(* IEC 61131-3 sources: types/src (part 2) *)

   END_TYPE

   TYPE EMHFDataRec147V1 : STRUCT
         version  : Byte := BYTE#1;   // Version
         resb1  : Byte;   // Reserved
         qualifierL1  : Word;   // Qualifier L1
         voltL1N  : Real;   // Voltage L1-N
         currentL1  : Real;   // Current L1
         apparentPowerL1  : Real;   // Apparent power L1
         activePowerL1  : Real;   // Active power L1
         reactivePowerQtotL1  : Real;   // Reactive power Qtot L1
         powerFactorL1  : Real;   // Power factor λ L1
         phaseAngleL1  : Real;   // Phase angle L1
         apparentEnergyLongL1  : LReal;   // Apparent energy L1
         totalActiveEnergyLongL1  : LReal;   // Active energy (total) L1
         totalReactiveEnergyLongL1  : LReal;   // Reactive energy (total) L1
         maxVoltL1N  : Real;   // Max. voltage L1-N
         maxCurrentL1  : Real;   // Max. current L1
         maxApparentPowerL1  : Real;   // Max. apparent power L1
         maxActivePowerL1  : Real;   // Max. active power L1
         maxReactivePowerQtotL1  : Real;   // Max. reactive power Qtot L1
         maxPowerFactorL1  : Real;   // Max. power factor λ L1
         minVoltL1N  : Real;   // Min. voltage L1-N
         minCurrentL1  : Real;   // Min. current L1
         minApparentPowerL1  : Real;   // Min. apparent power L1
         minActivePowerL1  : Real;   // Min. active power L1
         minReactivePowerQtotL1  : Real;   // Min. reactive power Qtot L1
         minPowerFactorL1  : Real;   // Min. power factor λ L1
         reactivePowerQnL1  : Real;   // Reactive power Qn L1
         voltL1Cycles10to12  : Real;   // Voltage L1 10-12 cycles
         currL1Cycles10to12  : Real;   // Current L1 10-12 cycles
         maxReactivePowerQnL1  : Real;   // Max. reactive power Qn L1
         minReactivePowerQnL1  : Real;   // Min. reactive power Qn L1
         fundVoltL1  : Real;   // Fundamental voltage L1
         fundCurrL1  : Real;   // Fundamental current L1
         fundApparentPowerL1  : Real;   // Fundamental apparent power L1
         fundReactivePowerL1  : Real;   // Fundamental reactive power L1
         fundActivePowerL1  : Real;   // Fundamental active power L1
         fundActiveFactorL1  : Real;   // Fundamental cos φ active factor L1
         maxFundVoltL1  : Real;   // Max. fundamental voltage L1
         maxFundCurrL1  : Real;   // Max. fundamental current L1
         maxFundApparentPowerL1  : Real;   // Max. fundamental apparent power L1
         maxFundReactivePowerL1  : Real;   // Max. fundamental reactive power L1
         maxFundActivePowerL1  : Real;   // Max. fundamental active power L1
         maxFundActiveFactorL1  : Real;   // Max. fundamental cos φ active factor L1
         minFundVoltL1  : Real;   // Min. fundamental voltage L1
         minFundCurrL1  : Real;   // Min. fundamental current L1
         minFundApparentPowerL1  : Real;   // Min. fundamental apparent power L1
         minFundReactivePowerL1  : Real;   // Min. fundamental reactive power L1
         minFundActivePowerL1  : Real;   // Min. fundamental active power L1
         minFundActiveFactorL1  : Real;   // Min. fundamental cos φ active factor L1
         tHDaNVoltL1  : Real;   // Total harmonic distortion (THD+N) voltage L1
         tHDaNCurrL1  : Real;   // Total harmonic distortion (THD+N) current L1
         maxTHDaNVoltL1  : Real;   // Max. total harmonic distortion (THD+N) voltage L1
         maxTHDaNCurrL1  : Real;   // Max. total harmonic distortion (THD+N) current L1
         minTHDaNVoltL1  : Real;   // Min. total harmonic distortion (THD+N) voltage L1
         minTHDaNCurrL1  : Real;   // Min. total harmonic distortion (THD+N) current L1
         voltDipValueL1  : Real;   // Voltage dip - value L1
         voltDipDurationL1  : Real;   // Voltage dip - duration L1
         voltSwellValueL1  : Real;   // Voltage swell - value L1
         voltSwellDurationL1  : Real;   // Voltage swell - duration L1
         voltPeakValueL1  : Real;   // Voltage peak value L1
         currPeakValueL1  : Real;   // Current peak value L1
         overCurrValueL1  : Real;   // Overcurrent value L1
      END_STRUCT;

   END_TYPE

   TYPE EMHFDataRec142V2 : STRUCT
         version  : Byte := BYTE#2;   // Version
         resb1  : Byte;   // Reserved
         voltL1N  : Real;   // Voltage L1-N
         voltL2N  : Real;   // Voltage L2-N
         voltL3N  : Real;   // Voltage L3-N
         voltL1L2  : Real;   // Voltage L1-L2
         voltL2L3  : Real;   // Voltage L2-L3
         voltL3L1  : Real;   // Voltage L3-L1
         currentL1  : Real;   // Current L1
         currentL2  : Real;   // Current L2
         currentL3  : Real;   // Current L3
         powerFactorL1  : Real;   // Power factor λ L1
         powerFactorL2  : Real;   // Power factor λ L2
         powerFactorL3  : Real;   // Power factor λ L3
         powerFactorL1L2L3  : Real;   // Power factor λ L1 L2 L3
         frequencyL1L2L3  : Real;   // Frequency L1 L2 L3
         amplUnbalanceVolt  : Real;   // Amplitude unbalance voltage U2
         amplUnbalanceCurrent  : Real;   // Amplitude unbalance current Iasym
         apparentPowerL1  : Real;   // Apparent power L1
         apparentPowerL2  : Real;   // Apparent power L2
         apparentPowerL3  : Real;   // Apparent power L3
         apparentPowerL1L2L3  : Real;   // Apparent power L1 L2 L3
         reactivePowerQtotL1  : Real;   // Reactive power Qtot L1
         reactivePowerQtotL2  : Real;   // Reactive power Qtot L2
         reactivePowerQtotL3  : Real;   // Reactive power Qtot L3
         reactivePowerQtotL1L2L3  : Real;   // Reactive power Qtot L1 L2 L3
         activePowerL1  : Real;   // Active power L1
         activePowerL2  : Real;   // Active power L2
         activePowerL3  : Real;   // Active power L3
         activePowerL1L2L3  : Real;   // Active power L1 L2 L3
         phaseAngleL1  : Real;   // Phase angle L1
         phaseAngleL2  : Real;   // Phase angle L2
         phaseAngleL3  : Real;   // Phase angle L3
         apparentEnergyL1L2L3  : Real;   // Apparent energy L1 L2 L3
         totalReactiveEnergyL1L2L3  : Real;   // Total reactive energy L1 L2 L3
         totalActiveEnergyL1L2L3  : Real;   // Total active energy L1 L2 L3
         reactiveEnergyInL1L2L3  : Real;   // Reactive energy inflow L1 L2 L3
         reactiveEnergyOutL1L2L3  : Real;   // Reactive energy outflow L1 L2 L3
         activeEnergyInL1L2L3  : Real;   // Active energy inflow L1 L2 L3
         activeEnergyOutL1L2L3  : Real;   // Active energy outflow L1 L2 L3
         apparentEnergyLongL1L2L3  : LReal;   // Apparent energy L1 L2 L3
         totalReactiveEnergyLongL1L2L3  : LReal;   // Total reactive energy L1 L2 L3
         totalActiveEnergyLongL1L2L3  : LReal;   // Total active energy L1 L2 L3
         reactiveEnergyInLongL1L2L3  : LReal;   // Reactive energy inflow L1 L2 L3
         reactiveEnergyOutLongL1L2L3  : LReal;   // Reactive energy outflow L1 L2 L3
         activeEnergyInLongL1L2L3  : LReal;   // Active energy inflow L1 L2 L3
         activeEnergyOutLongL1L2L3  : LReal;   // Active energy outflow L1 L2 L3
         neutralCurrentIn  : Real;   // Neutral current IN
      END_STRUCT;

   END_TYPE

   TYPE EMHFDataRec148V1 : STRUCT
         version  : Byte := BYTE#1;   // Version
         resb1  : Byte;   // Reserved
         qualifierL2  : Word;   // Qualifier L2
         voltL2N  : Real;   // Voltage L2-N
         currentL2  : Real;   // Current L2
         apparentPowerL2  : Real;   // Apparent power L2
         activePowerL2  : Real;   // Active power L2
         reactivePowerQtotL2  : Real;   // Reactive power Qtot L2
         powerFactorL2  : Real;   // Power factor λ L2
         phaseAngleL2  : Real;   // Phase angle L2
         apparentEnergyLongL2  : LReal;   // Apparent energy L2
         totalActiveEnergyLongL2  : LReal;   // Active energy (total) L2
         totalReactiveEnergyLongL2  : LReal;   // Reactive energy (total) L2
         maxVoltL2N  : Real;   // Max. voltage L2-N
         maxCurrentL2  : Real;   // Max. current L2
         maxApparentPowerL2  : Real;   // Max. apparent power L2
         maxActivePowerL2  : Real;   // Max. active power L2
         maxReactivePowerQtotL2  : Real;   // Max. reactive power Qtot L2
         maxPowerFactorL2  : Real;   // Max. power factor λ L2
         minVoltL2N  : Real;   // Min. voltage L2-N
         minCurrentL2  : Real;   // Min. current L2
         minApparentPowerL2  : Real;   // Min. apparent power L2
         minActivePowerL2  : Real;   // Min. active power L2
         minReactivePowerQtotL2  : Real;   // Min. reactive power Qtot L2
         minPowerFactorL2  : Real;   // Min. power factor λ L2
         reactivePowerQnL2  : Real;   // Reactive power Qn L2
         voltL2Cycles10to12  : Real;   // Voltage L2 10-12 cycles
         currL2Cycles10to12  : Real;   // Current L2 10-12 cycles
         maxReactivePowerQnL2  : Real;   // Max. reactive power Qn L2
         minReactivePowerQnL2  : Real;   // Min. reactive power Qn L2
         fundVoltL2  : Real;   // Fundamental voltage L2
         fundCurrL2  : Real;   // Fundamental current L2
         fundApparentPowerL2  : Real;   // Fundamental apparent power L2
         fundReactivePowerL2  : Real;   // Fundamental reactive power L2
         fundActivePowerL2  : Real;   // Fundamental active power L2
         fundActiveFactorL2  : Real;   // Fundamental cos φ active factor L2
         maxFundVoltL2  : Real;   // Max. fundamental voltage L2
         maxFundCurrL2  : Real;   // Max. fundamental current L2
         maxFundApparentPowerL2  : Real;   // Max. fundamental apparent power L2
         maxFundReactivePowerL2  : Real;   // Max. fundamental reactive power L2
         maxFundActivePowerL2  : Real;   // Max. fundamental active power L2
         maxFundActiveFactorL2  : Real;   // Max. fundamental cos φ active factor L2
         minFundVoltL2  : Real;   // Min. fundamental voltage L2
         minFundCurrL2  : Real;   // Min. fundamental current L2
         minFundApparentPowerL2  : Real;   // Min. fundamental apparent power L2
         minFundReactivePowerL2  : Real;   // Min. fundamental reactive power L2
         minFundActivePowerL2  : Real;   // Min. fundamental active power L2
         minFundActiveFactorL2  : Real;   // Min. fundamental cos φ active factor L2
         tHDaNVoltL2  : Real;   // Total harmonic distortion (THD+N) voltage L2
         tHDaNCurrL2  : Real;   // Total harmonic distortion (THD+N) current L2
         maxTHDaNVoltL2  : Real;   // Max. total harmonic distortion (THD+N) voltage L2
         maxTHDaNCurrL2  : Real;   // Max. total harmonic distortion (THD+N) current L2
         minTHDaNVoltL2  : Real;   // Min. total harmonic distortion (THD+N) voltage L2
         minTHDaNCurrL2  : Real;   // Min. total harmonic distortion (THD+N) current L2
         voltDipValueL2  : Real;   // Voltage dip - value L2
         voltDipDurationL2  : Real;   // Voltage dip - duration L2
         voltSwellValueL2  : Real;   // Voltage swell - value L2
         voltSwellDurationL2  : Real;   // Voltage swell - duration L2
         voltPeakValueL2  : Real;   // Voltage peak value L2
         currPeakValueL2  : Real;   // Current peak value L2
         overCurrValueL2  : Real;   // Overcurrent value L2
      END_STRUCT;

   END_TYPE

   TYPE EMSTDataRec142V2 : STRUCT
         version  : Byte := BYTE#2;   // Version
         resb1  : Byte;   // Reserved
         voltL1N  : Real;   // Voltage L1-N
         voltL2N  : Real;   // Voltage L2-N
         voltL3N  : Real;   // Voltage L3-N
         voltL1L2  : Real;   // Voltage L1-L2
         voltL2L3  : Real;   // Voltage L2-L3
         voltL3L1  : Real;   // Voltage L3-L1
         currentL1  : Real;   // Current L1
         currentL2  : Real;   // Current L2
         currentL3  : Real;   // Current L3
         powerFactorL1  : Real;   // Power factor λ L1
         powerFactorL2  : Real;   // Power factor λ L2
         powerFactorL3  : Real;   // Power factor λ L3
         powerFactorL1L2L3  : Real;   // Power factor L1 L2 L3
         frequencyL1L2L3  : Real;   // Frequency L1 L2 L3
         amplUnbalanceVolt  : Real;   // Amplitude unbalance voltage U2
         amplUnbalanceCurrent  : Real;   // Amplitude unbalance current Iasym
         apparentPowerL1  : Real;   // Apparent power L1
         apparentPowerL2  : Real;   // Apparent power L2
         apparentPowerL3  : Real;   // Apparent power L3
         apparentPowerL1L2L3  : Real;   // Apparent power L1 L2 L3
         reactivePowerQtotL1  : Real;   // Reactive power Qtot L1
         reactivePowerQtotL2  : Real;   // Reactive power Qtot L2
         reactivePowerQtotL3  : Real;   // Reactive power Qtot L3
         reactivePowerQtotL1L2L3  : Real;   // Reactive power Qtot L1 L2 L3
         activePowerL1  : Real;   // Active power L1
         activePowerL2  : Real;   // Active power L2
         activePowerL3  : Real;   // Active power L3
         activePowerL1L2L3  : Real;   // Active power L1 L2 L3
         phaseAngleL1  : Real;   // Phase angle L1
         phaseAngleL2  : Real;   // Phase angle L2
         phaseAngleL3  : Real;   // Phase angle L3
         apparentEnergyL1L2L3  : Real;   // Apparent energy L1 L2 L3
         totalReactiveEnergyL1L2L3  : Real;   // Total reactive energy L1 L2 L3
         totalActiveEnergyL1L2L3  : Real;   // Total active energy L1 L2 L3
         reactiveEnergyInL1L2L3  : Real;   // Reactive energy inflow L1 L2 L3
         reactiveEnergyOutL1L2L3  : Real;   // Reactive energy outflow L1 L2 L3
         activeEnergyInL1L2L3  : Real;   // Active energy inflow L1 L2 L3
         activeEnergyOutL1L2L3  : Real;   // Active energy outflow L1 L2 L3
         apparentEnergyLongL1L2L3  : LReal;   // Apparent energy L1 L2 L3
         totalReactiveEnergyLongL1L2L3  : LReal;   // Total reactive energy L1 L2 L3
         totalActiveEnergyLongL1L2L3  : LReal;   // Total active energy L1 L2 L3
         reactiveEnergyInLongL1L2L3  : LReal;   // Reactive energy inflow L1 L2 L3
         reactiveEnergyOutLongL1L2L3  : LReal;   // Reactive energy outflow L1 L2 L3
         activeEnergyInLongL1L2L3  : LReal;   // Active energy inflow L1 L2 L3
         activeEnergyOutLongL1L2L3  : LReal;   // Active energy outflow L1 L2 L3
         neutralCurrentIn  : Real;   // Neutral current IN
      END_STRUCT;

   END_TYPE

   TYPE EMHFDataRec154 : STRUCT
         version  : Byte := BYTE#2;   // Version
         resb1  : Byte;   // Reserved
         maxVoltL1N  : RealValueAndPNIOTimeStamp;   // Max. voltage L1-N
         maxVoltL2N  : RealValueAndPNIOTimeStamp;   // Max. voltage L2-N
         maxVoltL3N  : RealValueAndPNIOTimeStamp;   // Max. voltage L3-N
         maxVoltL1L2  : RealValueAndPNIOTimeStamp;   // Max. voltage L1-L2
         maxVoltL2L3  : RealValueAndPNIOTimeStamp;   // Max. voltage L2-L3
         maxVoltL3L1  : RealValueAndPNIOTimeStamp;   // Max. voltage L3-L1
         maxCurrentL1  : RealValueAndPNIOTimeStamp;   // Max. current L1
         maxCurrentL2  : RealValueAndPNIOTimeStamp;   // Max. current L2
         maxCurrentL3  : RealValueAndPNIOTimeStamp;   // Max. current L3
         maxApparentPowerL1  : RealValueAndPNIOTimeStamp;   // Max. apparent power L1
         maxApparentPowerL2  : RealValueAndPNIOTimeStamp;   // Max. apparent power L2
         maxApparentPowerL3  : RealValueAndPNIOTimeStamp;   // Max. apparent power L3
         maxActivePowerL1  : RealValueAndPNIOTimeStamp;   // Max. active power L1
         maxActivePowerL2  : RealValueAndPNIOTimeStamp;   // Max. active power L2
         maxActivePowerL3  : RealValueAndPNIOTimeStamp;   // Max. active power L3
         maxReactivePowerQtotL1  : RealValueAndPNIOTimeStamp;   // Max. reactive power Qtot L1
         maxReactivePowerQtotL2  : RealValueAndPNIOTimeStamp;   // Max. reactive power Qtot L2
         maxReactivePowerQtotL3  : RealValueAndPNIOTimeStamp;   // Max. reactive power Qtot L3
         maxPowerFactorL1  : RealValueAndPNIOTimeStamp;   // Max. power factor λ L1
         maxPowerFactorL2  : RealValueAndPNIOTimeStamp;   // Max. power factor λ L2
         maxPowerFactorL3  : RealValueAndPNIOTimeStamp;   // Max. power factor λ L3
         maxFrequency  : RealValueAndPNIOTimeStamp;   // Max. frequency
         maxApparentPowerL1L2L3  : RealValueAndPNIOTimeStamp;   // Max. apparent power L1 L2 L3
         maxActivePowerL1L2L3  : RealValueAndPNIOTimeStamp;   // Max. active power L1 L2 L3
         maxReactivePowerQtotL1L2L3  : RealValueAndPNIOTimeStamp;   // Max. reactive power Qtot L1 L2 L3
         maxPowerFactorL1L2L3  : RealValueAndPNIOTimeStamp;   // Max. power factor λ L1L2L3
         maxReactivePowerQnL1  : RealValueAndPNIOTimeStamp;   // Max. reactive power Qn L1
         maxReactivePowerQnL2  : RealValueAndPNIOTimeStamp;   // Max. reactive power Qn L2
         maxReactivePowerQnL3  : RealValueAndPNIOTimeStamp;   // Max. reactive power Qn L3
         maxMeanVoltLN  : RealValueAndPNIOTimeStamp;   // Max. mean voltage L-N
         maxMeanVoltLL  : RealValueAndPNIOTimeStamp;   // Max. mean voltage L-L
         maxSumMeanCurrL1L2L3  : RealValueAndPNIOTimeStamp;   // Max. sum mean value current L1L2L3
         maxFundVoltL1  : RealValueAndPNIOTimeStamp;   // Max. fundamental voltage L1
         maxFundVoltL2  : RealValueAndPNIOTimeStamp;   // Max. fundamental voltage L2
         maxFundVoltL3  : RealValueAndPNIOTimeStamp;   // Max. fundamental voltage L3
         maxFundCurrL1  : RealValueAndPNIOTimeStamp;   // Max. fundamental current L1
         maxFundCurrL2  : RealValueAndPNIOTimeStamp;   // Max. fundamental current L2
         maxFundCurrL3  : RealValueAndPNIOTimeStamp;   // Max. fundamental current L3
         maxFundApparentPowerL1  : RealValueAndPNIOTimeStamp;   // Max. fundamental apparent power L1
         maxFundApparentPowerL2  : RealValueAndPNIOTimeStamp;   // Max. fundamental apparent power L2
         maxFundApparentPowerL3  : RealValueAndPNIOTimeStamp;   // Max. fundamental apparent power L3
         maxFundReactivePowerL1  : RealValueAndPNIOTimeStamp;   // Max. fundamental reactive power L1
         maxFundReactivePowerL2  : RealValueAndPNIOTimeStamp;   // Max. fundamental reactive power L2
         maxFundReactivePowerL3  : RealValueAndPNIOTimeStamp;   // Max. fundamental reactive power L3
         maxFundActivePowerL1  : RealValueAndPNIOTimeStamp;   // Max. fundamental active power L1
         maxFundActivePowerL2  : RealValueAndPNIOTimeStamp;   // Max. fundamental active power L2
         maxFundActivePowerL3  : RealValueAndPNIOTimeStamp;   // Max. fundamental active power L3
         maxFundActiveFactorL1  : RealValueAndPNIOTimeStamp;   // Max. fundamental cos φ active factor L1
         maxFundActiveFactorL2  : RealValueAndPNIOTimeStamp;   // Max. fundamental cos φ active factor L2
         maxFundActiveFactorL3  : RealValueAndPNIOTimeStamp;   // Max. fundamental cos φ active factor L3
         maxTHDaNVoltL1  : RealValueAndPNIOTimeStamp;   // Max. total harmonic distortion (THD+N) voltage L1
         maxTHDaNVoltL2  : RealValueAndPNIOTimeStamp;   // Max. total harmonic distortion (THD+N) voltage L2
         maxTHDaNVoltL3  : RealValueAndPNIOTimeStamp;   // Max. total harmonic distortion (THD+N) voltage L3
         maxTHDaNCurrL1  : RealValueAndPNIOTimeStamp;   // Max. total harmonic distortion (THD+N) current L1
         maxTHDaNCurrL2  : RealValueAndPNIOTimeStamp;   // Max. total harmonic distortion (THD+N) current L2
         maxTHDaNCurrL3  : RealValueAndPNIOTimeStamp;   // Max. total harmonic distortion (THD+N) current L3
         maxNeutralCurr  : RealValueAndPNIOTimeStamp;   // Max. neutral current
      END_STRUCT;

   END_TYPE

   TYPE EMSTDataRec143 : STRUCT
         version  : Byte := BYTE#1;   // Version
         resb1  : Byte;   // Reserved
         controlStatusByte1L1  : Byte;   // Status / control byte 1 - L1
         controlStatusByte2L1  : Byte;   // Status / control byte 2 - L1
         controlStatusByte1L2  : Byte;   // Status / control byte 1 - L2
         controlStatusByte2L2  : Byte;   // Status / control byte 2 - L2
         controlStatusByte1L3  : Byte;   // Status / control byte 1 - L3
         controlStatusByte2L3  : Byte;   // Status / control byte 2 - L3
         activeEnergyInLongL1  : LReal;   // Active energy inflow (initial value) L1
         activeEnergyOutLongL1  : LReal;   // Active energy outflow (initial value) L1
         reactiveEnergyInLongL1  : LReal;   // Reactive energy inflow (initial value) L1
         reactiveEnergyOutLongL1  : LReal;   // Reactive energy outflow (initial value) L1
         apparentEnergyLongL1  : LReal;   // Apparent energy (initial value) L1
         activeEnergyInLongL2  : LReal;   // Active energy inflow (initial value) L2
         activeEnergyOutLongL2  : LReal;   // Active energy outflow (initial value) L2
         reactiveEnergyInLongL2  : LReal;   // Reactive energy inflow (initial value) L2
         reactiveEnergyOutLongL2  : LReal;   // Reactive energy outflow (initial value) L2
         apparentEnergyLongL2  : LReal;   // Apparent energy (initial value) L2
         activeEnergyInLongL3  : LReal;   // Active energy inflow (initial value) L3
         activeEnergyOutLongL3  : LReal;   // Active energy outflow (initial value) L3
         reactiveEnergyInLongL3  : LReal;   // Reactive energy inflow (initial value) L3
         reactiveEnergyOutLongL3  : LReal;   // Reactive energy outflow (initial value) L3
         apparentEnergyLongL3  : LReal;   // Apparent energy (initial value) L3
         ovCntActiveEnergyInL1  : UInt;   // Overflow counter active energy inflow L1
         ovCntActiveEnergyOutL1  : UInt;   // Overflow counter active energy outflow L1
         ovCntReactiveEnergyInL1  : UInt;   // Overflow counter reactive energy inflow L1
         ovCntReactiveEnergyOutL1  : UInt;   // Overflow counter reactive energy outflow L1
         ovCntApparentEnergyL1  : UInt;   // Overflow counter apparent energy L1
         ovCntActiveEnergyInL2  : UInt;   // Overflow counter active energy inflow L2
         ovCntActiveEnergyOutL2  : UInt;   // Overflow counter active energy outflow L2
         ovCntReactiveEnergyInL2  : UInt;   // Overflow counter reactive energy inflow L2
         ovCntReactiveEnergyOutL2  : UInt;   // Overflow counter reactive energy outflow L2
         ovCntApparentEnergyL2  : UInt;   // Overflow counter apparent energy L2
         ovCntActiveEnergyInL3  : UInt;   // Overflow counter active energy inflow L3
         ovCntActiveEnergyOutL3  : UInt;   // Overflow counter active energy outflow L3
         ovCntReactiveEnergyInL3  : UInt;   // Overflow counter reactive energy inflow L3
         ovCntReactiveEnergyOutL3  : UInt;   // Overflow counter reactive energy outflow L3
         ovCntApparentEnergyL3  : UInt;   // Overflow counter apparent energy L3
         operHoursCntL1  : Real;   // Operating hours counter L1 (initial value)
         operHoursCntL2  : Real;   // Operating hours counter L2 (initial value)
         operHoursCntL3  : Real;   // Operating hours counter L3 (initial value)
      END_STRUCT;

   END_TYPE

   TYPE EMSTDataRec135 : STRUCT
         majMinVer  : Byte := BYTE#0;   // Major / minor version
         dataRecordNum  : Byte := BYTE#151;   // Data record number for data record mapping = 151
         numMeasValues  : Byte := BYTE#150;   // Number of measured values for data record mapping
         resb3  : Byte;   // Reserved
         measValueID  : Array[1..150] of Word;   // ID of measured value for data record mapping
      END_STRUCT;

   END_TYPE

   TYPE EMHFDataRec149V1 : STRUCT
         version  : Byte := BYTE#1;   // Version
         resb1  : Byte;   // Reserved
         qualifierL3  : Word;   // Qualifier L3
         voltL3N  : Real;   // Voltage L3-N
         currentL3  : Real;   // Current L3
         apparentPowerL3  : Real;   // Apparent power L3
         activePowerL3  : Real;   // Active power L3
         reactivePowerQtotL3  : Real;   // Reactive power Qtot L3
         powerFactorL3  : Real;   // Power factor λ L3
         phaseAngleL3  : Real;   // Phase angle L3
         apparentEnergyLongL3  : LReal;   // Apparent energy L3
         totalActiveEnergyLongL3  : LReal;   // Active energy (total) L3
         totalReactiveEnergyLongL3  : LReal;   // Reactive energy (total) L3
         maxVoltL3N  : Real;   // Max. voltage L3-N
         maxCurrentL3  : Real;   // Max. current L3
         maxApparentPowerL3  : Real;   // Max. apparent power L3
         maxActivePowerL3  : Real;   // Max. active power L3
         maxReactivePowerQtotL3  : Real;   // Max. reactive power Qtot L3
         maxPowerFactorL3  : Real;   // Max. power factor λ L3
         minVoltL3N  : Real;   // Min. voltage L3-N
         minCurrentL3  : Real;   // Min. current L3
         minApparentPowerL3  : Real;   // Min. apparent power L3
         minActivePowerL3  : Real;   // Min. active power L3
         minReactivePowerQtotL3  : Real;   // Min. reactive power Qtot L3
         minPowerFactorL3  : Real;   // Min. power factor λ L3
         reactivePowerQnL3  : Real;   // Reactive power Qn L3
         voltL3Cycles10to12  : Real;   // Voltage L3 10-12 cycles
         currL3Cycles10to12  : Real;   // Current L3 10-12 cycles
         maxReactivePowerQnL3  : Real;   // Max. reactive power Qn L3
         minReactivePowerQnL3  : Real;   // Min. reactive power Qn L3
         fundVoltL3  : Real;   // Fundamental voltage L3
         fundCurrL3  : Real;   // Fundamental current L3
         fundApparentPowerL3  : Real;   // Fundamental apparent power L3
         fundReactivePowerL3  : Real;   // Fundamental reactive power L3
         fundActivePowerL3  : Real;   // Fundamental active power L3
         fundActiveFactorL3  : Real;   // Fundamental cos φ active factor L3
         maxFundVoltL3  : Real;   // Max. fundamental voltage L3
         maxFundCurrL3  : Real;   // Max. fundamental current L3
         maxFundApparentPowerL3  : Real;   // Max. fundamental apparent power L3
         maxFundReactivePowerL3  : Real;   // Max. fundamental reactive power L3
         maxFundActivePowerL3  : Real;   // Max. fundamental active power L3
         maxFundActiveFactorL3  : Real;   // Max. fundamental cos φ active factor L3
         minFundVoltL3  : Real;   // Min. fundamental voltage L3
         minFundCurrL3  : Real;   // Min. fundamental current L3
         minFundApparentPowerL3  : Real;   // Min. fundamental apparent power L3
         minFundReactivePowerL3  : Real;   // Min. fundamental reactive power L3
         minFundActivePowerL3  : Real;   // Min. fundamental active power L3
         minFundActiveFactorL3  : Real;   // Min. fundamental cos φ active factor L3
         tHDaNVoltL3  : Real;   // Total harmonic distortion (THD+N) voltage L3
         tHDaNCurrL3  : Real;   // Total harmonic distortion (THD+N) current L3
         maxTHDaNVoltL3  : Real;   // Max. total harmonic distortion (THD+N) voltage L3
         maxTHDaNCurrL3  : Real;   // Max. total harmonic distortion (THD+N) current L3
         minTHDaNVoltL3  : Real;   // Min. total harmonic distortion (THD+N) voltage L3
         minTHDaNCurrL3  : Real;   // Min. total harmonic distortion (THD+N) current L3
         voltDipValueL3  : Real;   // Voltage dip - value L3
         voltDipDurationL3  : Real;   // Voltage dip - duration L3
         voltSwellValueL3  : Real;   // Voltage swell - value L3
         voltSwellDurationL3  : Real;   // Voltage swell - duration L3
         voltPeakValueL3  : Real;   // Voltage peak value L3
         currPeakValueL3  : Real;   // Current peak value L3
         overCurrValueL3  : Real;   // Overcurrent value L3
      END_STRUCT;

   END_TYPE

   TYPE EMHFDataRec150V1 : STRUCT
         version  : Byte := BYTE#1;   // Version
         resb1  : Byte;   // Reserved
         operHoursCntL1L2L3  : Real;   // Operating hours counter L1 L2 L3
         operHoursCntL1  : Real;   // Operating hours counter L1
         operHoursCntL2  : Real;   // Operating hours counter L2
         operHoursCntL3  : Real;   // Operating hours counter L3
         statusLimViolGW1to16  : Word;   // Status limit violation GW 1...16
         statusEnergyCntOv  : Word;   // Status of energy counter overflows
         cntLimViolGw1  : UDInt;   // Counter limit violation GW 1
         cntLimViolGw2  : UDInt;   // Counter limit violation GW 2
         cntLimViolGw3  : UDInt;   // Counter limit violation GW 3
         cntLimViolGw4  : UDInt;   // Counter limit violation GW 4
         cntLimViolGw5  : UDInt;   // Counter limit violation GW 5
         cntLimViolGw6  : UDInt;   // Counter limit violation GW 6
         cntLimViolGw7  : UDInt;   // Counter limit violation GW 7
         cntLimViolGw8  : UDInt;   // Counter limit violation GW 8
         cntLimViolGw9  : UDInt;   // Counter limit violation GW 9
         cntLimViolGw10  : UDInt;   // Counter limit violation GW 10
         cntLimViolGw11  : UDInt;   // Counter limit violation GW 11
         cntLimViolGw12  : UDInt;   // Counter limit violation GW 12
         cntLimViolGw13  : UDInt;   // Counter limit violation GW 13
         cntLimViolGw14  : UDInt;   // Counter limit violation GW 14
         cntLimViolGw15  : UDInt;   // Counter limit violation GW 15
         cntLimViolGw16  : UDInt;   // Counter limit violation GW 16
         qualifierL1L2L3  : Word;   // Qualifier L1 L2 L3
         powerQualityAnalysis  : UDInt;   // Power quality analysis - Qualifier
         currentModuleTime  : PNIOTimeStamp;   // Current module time
      END_STRUCT;

   END_TYPE

   TYPE TMTimerDIDQ10DataRec : STRUCT
         majMinVer  : Byte := BYTE#1;   // Major / minor version
         channelParamLength  : Byte := BYTE#36;   // Length of the parameter data = 36
         reserved0  : Word;   // Reserved
         pwmPeriod  : Byte;   // Reserved/ PWM period for the digital outputs
         enableDiagnostics  : Byte;   // Enable diagnostics / Reaction to CPU STOP
         reserved1  : Word;   // Reserved
         operatingModeDI0  : Byte;   // Reserved / invert input signal / operating mode DI0
         inputDelayDI0  : Byte;   // Reserved / Input delay / Filter frequency DI0
         operatingModeDI1  : Byte;   // Reserved / invert input signal / operating mode DI1
         inputDelayDI1  : Byte;   // Reserved / Input delay / Filter frequency DI1
         operatingModeDI2  : Byte;   // Reserved / invert input signal / HW enable with DI3 / operating mode DI2
         inputDelayDI2  : Byte;   // Reserved / Input delay / Filter frequency DI2
         operatingModeDI3  : Byte;   // Reserved / invert input signal / operating mode DI1
         inputDelayDI3  : Byte;   // Reserved / Input delay DI3
         operatingModeDQ0  : Byte;   // High-speed output / Substitute value / invert input signal / HW enable / operating mode DQ0
         reserved2  : Byte;   // Reserved
         operatingModeDQ1  : Byte;   // High-speed output / Substitute value / invert input signal / HW enable / operating mode DQ1
         reserved3  : Byte;   // Reserved
         operatingModeDQ2  : Byte;   // High-speed output / Substitute value / invert input signal / HW enable / operating mode DQ2
         reserved4  : Byte;   // Reserved
         operatingModeDQ3  : Byte;   // High-speed output / Substitute value / invert input signal / Reserved / operating mode DQ3
         reserved5  : Byte;   // Reserved
         operatingModeDQ4  : Byte;   // High-speed output / Substitute value / invert input signal / Reserved / operating mode DQ4
         reserved6  : Byte;   // Reserved
         operatingModeDQ5  : Byte;   // High-speed output / Substitute value / invert input signal / Reserved / operating mode DQ5
         reserved7  : Byte;   // Reserved
         reserved8  : DWord;   // Reserved
         reserved9  : DWord;   // Reserved
         reserved10  : DWord;   // Reserved
      END_STRUCT;

   END_TYPE

   TYPE EMSTDataRec130 : STRUCT
         majMinVer  : Byte := BYTE#0;   // Major / minor version
         numUserDataVariant  : Byte := BYTE#1;   // Number of user data variant = 1
         numMeasValues  : Byte;   // Number of measured values for payload mapping
         resb3  : Byte;   // Reserved
         measValue  : Array[1..64] of Word;   // ID of measured value for payload mapping
      END_STRUCT;

   END_TYPE

   TYPE EMSTDataRec148V1 : STRUCT
         version  : Byte := BYTE#1;   // Version
         resb1  : Byte;   // Reserved
         qualifierL2  : Word;   // Qualifier L2
         voltL2N  : Real;   // Voltage L2-N
         currentL2  : Real;   // Current L2
         apparentPowerL2  : Real;   // Apparent power L2
         activePowerL2  : Real;   // Active power L2
         reactivePowerQtotL2  : Real;   // Reactive power Qtot L2
         powerFactorL2  : Real;   // Power factor λ L2
         phaseAngleL2  : Real;   // Phase angle L2
         apparentEnergyLongL2  : LReal;   // Apparent energy L2
         totalActiveEnergyLongL2  : LReal;   // Active energy (total) L2
         totalReactiveEnergyLongL2  : LReal;   // Reactive energy (total) L2
         maxVoltL2N  : Real;   // Max. voltage L2-N
         maxCurrentL2  : Real;   // Max. current L2
         maxApparentPowerL2  : Real;   // Max. apparent power L2
         maxActivePowerL2  : Real;   // Max. active power L2
         maxReactivePowerQtotL2  : Real;   // Max. reactive power Qtot L2
         maxPowerFactorL2  : Real;   // Max. power factor λ L2
         minVoltL2N  : Real;   // Min. voltage L2-N
         minCurrentL2  : Real;   // Min. current L2
         minApparentPowerL2  : Real;   // Min. apparent power L2
         minActivePowerL2  : Real;   // Min. active power L2
         minReactivePowerQtotL2  : Real;   // Min. reactive power Qtot L2
         minPowerFactorL2  : Real;   // Min. power factor λ L2
         reactivePowerQnL2  : Real;   // Reactive power Qn L2
         resDW108  : DWord;   // Reserved
         resDW112  : Real;   // Reserved
         resDW116  : Real;   // Reserved
         resDW120  : Real;   // Reserved
         resDW124  : Real;   // Reserved
         resDW128  : Real;   // Reserved
         resDW132  : Real;   // Reserved
         fundReactivePowerL2  : Real;   // Fundamental reactive power L2
         resDW140  : DWord;   // Reserved
         fundActiveFactorL2  : Real;   // Fundamental cos φ active factor L2
         resDW148  : DWord;   // Reserved
         resDW152  : DWord;   // Reserved
         resDW156  : DWord;   // Reserved
         resDW160  : DWord;   // Reserved
         resDW164  : DWord;   // Reserved
         resDW168  : DWord;   // Reserved
         resDW172  : DWord;   // Reserved
         resDW176  : DWord;   // Reserved
         resDW180  : DWord;   // Reserved
         resDW184  : DWord;   // Reserved
         resDW188  : DWord;   // Reserved
         resDW192  : DWord;   // Reserved
         resDW196  : DWord;   // Reserved
         resDW200  : DWord;   // Reserved
         resDW204  : DWord;   // Reserved
         resDW208  : DWord;   // Reserved
         resDW212  : DWord;   // Reserved
         resDW216  : DWord;   // Reserved
         resDW220  : DWord;   // Reserved
         resDW224  : DWord;   // Reserved
         resDW228  : DWord;   // Reserved
         resDW232  : DWord;   // Reserved
         resDW236  : DWord;   // Reserved
         resDW240  : DWord;   // Reserved
         resDW244  : DWord;   // Reserved
      END_STRUCT;

   END_TYPE

   TYPE EMHFDataRec130a131 : STRUCT
         majMinVer  : Byte := BYTE#0;   // Major / minor version
         numPayloadVariant  : Byte;   // Number of payload variant 1 or 2
         numMeasValues  : Byte := BYTE#64;   // Number of measured values for payload mapping
         resb3  : Byte;   // Reserved
         measValue  : Array[1..64] of Word;   // ID of measured value for payload mapping
      END_STRUCT;

   END_TYPE

   TYPE EMHFDataRec155 : STRUCT
         version  : Byte := BYTE#2;   // Version
         resb1  : Byte;   // Reserved
         minVoltL1N  : RealValueAndPNIOTimeStamp;   // Min. voltage L1-N
         minVoltL2N  : RealValueAndPNIOTimeStamp;   // Min. voltage L2-N
         minVoltL3N  : RealValueAndPNIOTimeStamp;   // Min. voltage L3-N
         minVoltL1L2  : RealValueAndPNIOTimeStamp;   // Min. voltage L1-L2
         minVoltL2L3  : RealValueAndPNIOTimeStamp;   // Min. voltage L2-L3
         minVoltL3L1  : RealValueAndPNIOTimeStamp;   // Min. voltage L3-L1
         minCurrentL1  : RealValueAndPNIOTimeStamp;   // Min. current L1
         minCurrentL2  : RealValueAndPNIOTimeStamp;   // Min. current L2
         minCurrentL3  : RealValueAndPNIOTimeStamp;   // Min. current L3
         minApparentPowerL1  : RealValueAndPNIOTimeStamp;   // Min. apparent power L1
         minApparentPowerL2  : RealValueAndPNIOTimeStamp;   // Min. apparent power L2
         minApparentPowerL3  : RealValueAndPNIOTimeStamp;   // Min. apparent power L3
         minActivePowerL1  : RealValueAndPNIOTimeStamp;   // Min. active power L1
         minActivePowerL2  : RealValueAndPNIOTimeStamp;   // Min. active power L2
         minActivePowerL3  : RealValueAndPNIOTimeStamp;   // Min. active power L3
         minReactivePowerQtotL1  : RealValueAndPNIOTimeStamp;   // Min. reactive power Qtot L1
         minReactivePowerQtotL2  : RealValueAndPNIOTimeStamp;   // Min. reactive power Qtot L2
         minReactivePowerQtotL3  : RealValueAndPNIOTimeStamp;   // Min. reactive power Qtot L3
         minPowerFactorL1  : RealValueAndPNIOTimeStamp;   // Min. power factor λ L1
         minPowerFactorL2  : RealValueAndPNIOTimeStamp;   // Min. power factor λ L2
         minPowerFactorL3  : RealValueAndPNIOTimeStamp;   // Min. power factor λ L3
         minFrequency  : RealValueAndPNIOTimeStamp;   // Min. frequency
         minlApparentPowerL1L2L3  : RealValueAndPNIOTimeStamp;   // Min. apparent power L1 L2 L3
         minActivePowerL1L2L3  : RealValueAndPNIOTimeStamp;   // Min. active power L1 L2 L3
         minReactivePowerQnL1L2L3  : RealValueAndPNIOTimeStamp;   // Min. reactive power Qn L1 L2 L3
         minPowerFactorL1L2L3  : RealValueAndPNIOTimeStamp;   // Min. power factor λ L1 L2 L3
         minReactivePowerQnL1  : RealValueAndPNIOTimeStamp;   // Min. reactive power Qn L1
         minReactivePowerQnL2  : RealValueAndPNIOTimeStamp;   // Min. reactive power Qn L2
         minReactivePowerQnL3  : RealValueAndPNIOTimeStamp;   // Min. reactive power Qn L3
         minMeanVoltLN  : RealValueAndPNIOTimeStamp;   // Min. mean voltage L-N
         minMeanVoltLL  : RealValueAndPNIOTimeStamp;   // Min. mean voltage L-L
         minMeanCurrL1L2L3  : RealValueAndPNIOTimeStamp;   // Min. mean current L1 L2 L3
         minFundVoltL1  : RealValueAndPNIOTimeStamp;   // Min. fundamental voltage L1
         minFundVoltL2  : RealValueAndPNIOTimeStamp;   // Min. fundamental voltage L2
         minFundVoltL3  : RealValueAndPNIOTimeStamp;   // Min. fundamental voltage L3
         minFundCurrL1  : RealValueAndPNIOTimeStamp;   // Min. fundamental current L1
         minFundCurrL2  : RealValueAndPNIOTimeStamp;   // Min. fundamental current L2
         minFundCurrL3  : RealValueAndPNIOTimeStamp;   // Min. fundamental current L3
         minFundApparentPowerL1  : RealValueAndPNIOTimeStamp;   // Min. fundamental apparent power L1
         minFundApparentPowerL2  : RealValueAndPNIOTimeStamp;   // Min. fundamental apparent power L2
         minFundApparentPowerL3  : RealValueAndPNIOTimeStamp;   // Min. fundamental apparent power L3
         minFundReactivePowerL1  : RealValueAndPNIOTimeStamp;   // Min. fundamental reactive power L1
         minFundReactivePowerL2  : RealValueAndPNIOTimeStamp;   // Min. fundamental reactive power L2
         minFundReactivePowerL3  : RealValueAndPNIOTimeStamp;   // Min. fundamental reactive power L3
         minFundActivePowerL1  : RealValueAndPNIOTimeStamp;   // Min. fundamental active power L1
         minFundActivePowerL2  : RealValueAndPNIOTimeStamp;   // Min. fundamental active power L2
         minFundActivePowerL3  : RealValueAndPNIOTimeStamp;   // Min. fundamental active power L3
         minFundActiveFactorL1  : RealValueAndPNIOTimeStamp;   // Min. fundamental cos φ active factor L1
         minFundActiveFactorL2  : RealValueAndPNIOTimeStamp;   // Min. fundamental cos φ active factor L2
         minFundActiveFactorL3  : RealValueAndPNIOTimeStamp;   // Min. fundamental cos φ active factor L3
         minTHDaNVoltL1  : RealValueAndPNIOTimeStamp;   // Min. total harmonic distortion (THD+N) voltage L1
         minTHDaNVoltL2  : RealValueAndPNIOTimeStamp;   // Min. total harmonic distortion (THD+N) voltage L2
         minTHDaNVoltL3  : RealValueAndPNIOTimeStamp;   // Min. total harmonic distortion (THD+N) voltage L3
         minTHDaNCurrL1  : RealValueAndPNIOTimeStamp;   // Min. total harmonic distortion (THD+N) current L1
         minTHDaNCurrL2  : RealValueAndPNIOTimeStamp;   // Min. total harmonic distortion (THD+N) current L2
         minTHDaNCurrL3  : RealValueAndPNIOTimeStamp;   // Min. total harmonic distortion (THD+N) current L3
         minNeutralCurr  : RealValueAndPNIOTimeStamp;   // Min. neutral current
      END_STRUCT;

   END_TYPE

   TYPE EMSTDataRec155 : STRUCT
         version  : Byte := BYTE#2;   // Version
         resb1  : Byte;   // Reserved
         minVoltL1N  : RealValueAndPNIOTimeStamp;   // Min. voltage L1-N
         minVoltL2N  : RealValueAndPNIOTimeStamp;   // Min. voltage L2-N
         minVoltL3N  : RealValueAndPNIOTimeStamp;   // Min. voltage L3-N
         minVoltL1L2  : RealValueAndPNIOTimeStamp;   // Min. voltage L1-L2
         minVoltL2L3  : RealValueAndPNIOTimeStamp;   // Min. voltage L2-L3
         minVoltL3L1  : RealValueAndPNIOTimeStamp;   // Min. voltage L3-L1
         minCurrentL1  : RealValueAndPNIOTimeStamp;   // Min. current L1
         minCurrentL2  : RealValueAndPNIOTimeStamp;   // Min. current L2
         minCurrentL3  : RealValueAndPNIOTimeStamp;   // Min. current L3
         minApparentPowerL1  : RealValueAndPNIOTimeStamp;   // Min. apparent power L1
         minApparentPowerL2  : RealValueAndPNIOTimeStamp;   // Min. apparent power L2
         minApparentPowerL3  : RealValueAndPNIOTimeStamp;   // Min. apparent power L3
         minActivePowerL1  : RealValueAndPNIOTimeStamp;   // Min. active power L1
         minActivePowerL2  : RealValueAndPNIOTimeStamp;   // Min. active power L2
         minActivePowerL3  : RealValueAndPNIOTimeStamp;   // Min. active power L3
         minReactivePowerQtotL1  : RealValueAndPNIOTimeStamp;   // Min. reactive power Qtot L1
         minReactivePowerQtotL2  : RealValueAndPNIOTimeStamp;   // Min. reactive power Qtot L2
         minReactivePowerQtotL3  : RealValueAndPNIOTimeStamp;   // Min. reactive power Qtot L3
         minPowerFactorL1  : RealValueAndPNIOTimeStamp;   // Min. power factor λ L1
         minPowerFactorL2  : RealValueAndPNIOTimeStamp;   // Min. power factor λ L2
         minPowerFactorL3  : RealValueAndPNIOTimeStamp;   // Min. power factor λ L3
         minFrequency  : RealValueAndPNIOTimeStamp;   // Min. frequency
         minlApparentPowerL1L2L3  : RealValueAndPNIOTimeStamp;   // Min. apparent power L1 L2 L3
         minActivePowerL1L2L3  : RealValueAndPNIOTimeStamp;   // Min. active power L1 L2 L3
         minReactivePowerQnL1L2L3  : RealValueAndPNIOTimeStamp;   // Min. reactive power Qn L1 L2 L3
         minPowerFactorL1L2L3  : RealValueAndPNIOTimeStamp;   // Min. power factor λ L1 L2 L3
         minReactivePowerQnL1  : RealValueAndPNIOTimeStamp;   // Min. reactive power Qn L1
         minReactivePowerQnL2  : RealValueAndPNIOTimeStamp;   // Min. reactive power Qn L2
         minReactivePowerQnL3  : RealValueAndPNIOTimeStamp;   // Min. reactive power Qn L3
         resByteArray466  : Array[0..15] of Byte;   // Reserved
         resByteArray482  : Array[0..15] of Byte;   // Reserved
         resByteArray498  : Array[0..15] of Byte;   // Reserved
         resByteArray514  : Array[0..15] of Byte;   // Reserved
         resByteArray530  : Array[0..15] of Byte;   // Reserved
         resByteArray546  : Array[0..15] of Byte;   // Reserved
         resByteArray562  : Array[0..15] of Byte;   // Reserved
         resByteArray578  : Array[0..15] of Byte;   // Reserved
         resByteArray594  : Array[0..15] of Byte;   // Reserved
         resByteArray610  : Array[0..15] of Byte;   // Reserved
         resByteArray626  : Array[0..15] of Byte;   // Reserved
         resByteArray642  : Array[0..15] of Byte;   // Reserved
         resByteArray658  : Array[0..15] of Byte;   // Reserved
         resByteArray674  : Array[0..15] of Byte;   // Reserved
         resByteArray690  : Array[0..15] of Byte;   // Reserved
         resByteArray706  : Array[0..15] of Byte;   // Reserved
         resByteArray722  : Array[0..15] of Byte;   // Reserved
         resByteArray738  : Array[0..15] of Byte;   // Reserved
         resByteArray754  : Array[0..15] of Byte;   // Reserved
         resByteArray770  : Array[0..15] of Byte;   // Reserved
         resByteArray786  : Array[0..15] of Byte;   // Reserved
         resByteArray802  : Array[0..15] of Byte;   // Reserved
         resByteArray818  : Array[0..15] of Byte;   // Reserved
         resByteArray834  : Array[0..15] of Byte;   // Reserved
         resByteArray850  : Array[0..15] of Byte;   // Reserved
         resByteArray866  : Array[0..15] of Byte;   // Reserved
         resByteArray882  : Array[0..15] of Byte;   // Reserved
         minNeutralCurr  : RealValueAndPNIOTimeStamp;   // Min. neutral current
      END_STRUCT;

   END_TYPE

   TYPE EMHFDataRec134 : STRUCT
         lowHighVer  : Byte := BYTE#0;   // Version low / high
         numDataRecord  : Byte := BYTE#173;   // Data record number for recorded measured values
         numMeasValues  : Byte;   // Number of activated measured values recordings
         resb3  : Byte;   // Reserved
         measValueRecBlock  : Array[1..2] of EMHFMeasValRecBlock;   // ID of measured value for payload mapping
      END_STRUCT;

   END_TYPE

   TYPE EMSTDataRec154 : STRUCT
         version  : Byte := BYTE#2;   // Version
         resb1  : Byte;   // Reserved
         maxVoltL1N  : RealValueAndPNIOTimeStamp;   // Max. voltage L1-N
         maxVoltL2N  : RealValueAndPNIOTimeStamp;   // Max. voltage L2-N
         maxVoltL3N  : RealValueAndPNIOTimeStamp;   // Max. voltage L3-N
         maxVoltL1L2  : RealValueAndPNIOTimeStamp;   // Max. voltage L1-L2
         maxVoltL2L3  : RealValueAndPNIOTimeStamp;   // Max. voltage L2-L3
         maxVoltL3L1  : RealValueAndPNIOTimeStamp;   // Max. voltage L3-L1
         maxCurrentL1  : RealValueAndPNIOTimeStamp;   // Max. current L1
         maxCurrentL2  : RealValueAndPNIOTimeStamp;   // Max. current L2
         maxCurrentL3  : RealValueAndPNIOTimeStamp;   // Max. current L3
         maxApparentPowerL1  : RealValueAndPNIOTimeStamp;   // Max. apparent power L1
         maxApparentPowerL2  : RealValueAndPNIOTimeStamp;   // Max. apparent power L2
         maxApparentPowerL3  : RealValueAndPNIOTimeStamp;   // Max. apparent power L3
         maxActivePowerL1  : RealValueAndPNIOTimeStamp;   // Max. active power L1
         maxActivePowerL2  : RealValueAndPNIOTimeStamp;   // Max. active power L2
         maxActivePowerL3  : RealValueAndPNIOTimeStamp;   // Max. active power L3
         maxReactivePowerQtotL1  : RealValueAndPNIOTimeStamp;   // Max. reactive power Qtot L1
         maxReactivePowerQtotL2  : RealValueAndPNIOTimeStamp;   // Max. reactive power Qtot L2
         maxReactivePowerQtotL3  : RealValueAndPNIOTimeStamp;   // Max. reactive power Qtot L3
         maxPowerFactorL1  : RealValueAndPNIOTimeStamp;   // Max. power factor λ L1
         maxPowerFactorL2  : RealValueAndPNIOTimeStamp;   // Max. power factor λ L2
         maxPowerFactorL3  : RealValueAndPNIOTimeStamp;   // Max. power factor λ L3
         maxFrequency  : RealValueAndPNIOTimeStamp;   // Max. frequency
         maxApparentPowerL1L2L3  : RealValueAndPNIOTimeStamp;   // Max. apparent power L1 L2 L3
         maxActivePowerL1L2L3  : RealValueAndPNIOTimeStamp;   // Max. active power L1 L2 L3
         maxReactivePowerQtotL1L2L3  : RealValueAndPNIOTimeStamp;   // Max. reactive power Qtot L1 L2 L3
         maxPowerFactorL1L2L3  : RealValueAndPNIOTimeStamp;   // Max. power factor λ L1L2L3
         maxReactivePowerQnL1  : RealValueAndPNIOTimeStamp;   // Max. reactive power Qn L1
         maxReactivePowerQnL2  : RealValueAndPNIOTimeStamp;   // Max. reactive power Qn L2
         maxReactivePowerQnL3  : RealValueAndPNIOTimeStamp;   // Max. reactive power Qn L3
         resByteArray466  : Array[0..15] of Byte;   // Reserved
         resByteArray482  : Array[0..15] of Byte;   // Reserved
         resByteArray498  : Array[0..15] of Byte;   // Reserved
         resByteArray514  : Array[0..15] of Byte;   // Reserved
         resByteArray530  : Array[0..15] of Byte;   // Reserved
         resByteArray546  : Array[0..15] of Byte;   // Reserved
         resByteArray562  : Array[0..15] of Byte;   // Reserved
         resByteArray578  : Array[0..15] of Byte;   // Reserved
         resByteArray594  : Array[0..15] of Byte;   // Reserved
         resByteArray610  : Array[0..15] of Byte;   // Reserved
         resByteArray626  : Array[0..15] of Byte;   // Reserved
         resByteArray642  : Array[0..15] of Byte;   // Reserved
         resByteArray658  : Array[0..15] of Byte;   // Reserved
         resByteArray674  : Array[0..15] of Byte;   // Reserved
         resByteArray690  : Array[0..15] of Byte;   // Reserved
         resByteArray706  : Array[0..15] of Byte;   // Reserved
         resByteArray722  : Array[0..15] of Byte;   // Reserved
         resByteArray738  : Array[0..15] of Byte;   // Reserved
         resByteArray754  : Array[0..15] of Byte;   // Reserved
         resByteArray770  : Array[0..15] of Byte;   // Reserved
         resByteArray786  : Array[0..15] of Byte;   // Reserved
         resByteArray802  : Array[0..15] of Byte;   // Reserved
         resByteArray818  : Array[0..15] of Byte;   // Reserved
         resByteArray834  : Array[0..15] of Byte;   // Reserved
         resByteArray850  : Array[0..15] of Byte;   // Reserved
         resByteArray866  : Array[0..15] of Byte;   // Reserved
         resByteArray882  : Array[0..15] of Byte;   // Reserved
         maxNeutralCurr  : RealValueAndPNIOTimeStamp;   // Max. neutral current
      END_STRUCT;

   END_TYPE

   TYPE TMTimerDIDQ10Control : STRUCT
         setDQ0  : Bool;   // Set DQ0 in the DQ operating mode Timer DQ
         setDQ1  : Bool;   // Set DQ1 in the DQ operating mode Timer DQ
         setDQ2  : Bool;   // Set DQ2 in the DQ operating mode Timer DQ
         setDQ3  : Bool;   // Set DQ3 in the DQ operating mode Timer DQ
         setDQ4  : Bool;   // Set DQ4 in the DQ operating mode Timer DQ
         setDQ5  : Bool;   // Set DQ5 in the DQ operating mode Timer DQ
         reserved0  : Bool;   // Reserved
         reserved1  : Bool;   // Reserved
         setEnDI0  : Bool;   // Override hardware enable for DI0
         setEnDI1  : Bool;   // Override hardware enable for DI1
         setEnDI2  : Bool;   // Override hardware enable for DI2
         setEnDI3  : Bool;   // Override hardware enable for DI3
         setEnDQ0  : Bool;   // Override hardware enable for DQ0
         setEnDQ1  : Bool;   // Override hardware enable for DQ1
         setEnDQ2  : Bool;   // Override hardware enable for DQ2
         setEnDQ3  : Bool;   // Override hardware enable for DQ3
         setEnDQ4  : Bool;   // Override hardware enable for DQ4
         setEnDQ5  : Bool;   // Override hardware enable for DQ5
         reserved2  : Bool;   // Reserved
         reserved3  : Bool;   // Reserved
         reserved4  : Bool;   // Reserved
         reserved5  : Bool;   // Reserved
         reserved6  : Bool;   // Reserved
         reserved7  : Bool;   // Reserved
         reserved8  : Byte;   // Reserved
         tecOutDQ0  : DWord;   // Value depends on DQ operating mode
         tecOutDQ1  : DWord;   // Value depends on DQ operating mode
         tecOutDQ2  : DWord;   // Value depends on DQ operating mode
         tecOutDQ3  : DWord;   // Value depends on DQ operating mode
         tecOutDQ4  : DWord;   // Value depends on DQ operating mode
         tecOutDQ5  : DWord;   // Value depends on DQ operating mode
         selDI0  : Byte;   // This Value is supplied by the TIO instruction TIO_DI
         selDI2  : Byte;   // This Value is supplied by the TIO instruction TIO_DI
         stw  : Word;   // This Value is controlled by the TIO instruction TIO_SYNC
      END_STRUCT;

   END_TYPE

   TYPE EMSTDataRec151Real : STRUCT
         version  : Byte;   // Version
         numMeasValues  : Byte := BYTE#150;   // Number of measured values for data record mapping
         measValue  : Array[1..150] of Real;   // ID of measured value for user data mapping
      END_STRUCT;

   END_TYPE

   TYPE DI8HSOVS : STRUCT
         channel  : Array[0..7] of OVSCh;   // Output values channel 0..7 with oversampling
      END_STRUCT;

   END_TYPE

   TYPE EMSTDataRec150V1 : STRUCT
         version  : Byte := BYTE#1;   // Version
         resb1  : Byte;   // Reserved
         operHoursCntL1L2L3  : Real;   // Operating hours counter L1 L2 L3
         operHoursCntL1  : Real;   // Operating hours counter L1
         operHoursCntL2  : Real;   // Operating hours counter L2
         operHoursCntL3  : Real;   // Operating hours counter L3
         statusLimViolGW1to16  : Word;   // Status limit violation GW 1...16
         statusEnergyCntOv  : Word;   // Status of energy counter overflows
         cntLimViolGw1  : UDInt;   // Counter limit violation GW 1
         cntLimViolGw2  : UDInt;   // Counter limit violation GW 2
         cntLimViolGw3  : UDInt;   // Counter limit violation GW 3
         cntLimViolGw4  : UDInt;   // Counter limit violation GW 4
         cntLimViolGw5  : UDInt;   // Counter limit violation GW 5
         cntLimViolGw6  : UDInt;   // Counter limit violation GW 6
         cntLimViolGw7  : UDInt;   // Counter limit violation GW 7
         cntLimViolGw8  : UDInt;   // Counter limit violation GW 8
         cntLimViolGw9  : UDInt;   // Counter limit violation GW 9
         cntLimViolGw10  : UDInt;   // Counter limit violation GW 10
         cntLimViolGw11  : UDInt;   // Counter limit violation GW 11
         cntLimViolGw12  : UDInt;   // Counter limit violation GW 12
         cntLimViolGw13  : UDInt;   // Counter limit violation GW 13
         cntLimViolGw14  : UDInt;   // Counter limit violation GW 14
         cntLimViolGw15  : UDInt;   // Counter limit violation GW 15
         cntLimViolGw16  : UDInt;   // Counter limit violation GW 16
         qualifierL1L2L3  : Word;   // Qualifier L1 L2 L3
         resUDINT88  : UDInt;   // Reserved
         currentModuleTime  : PNIOTimeStamp;   // Current module time
      END_STRUCT;

   END_TYPE

   TYPE EMHFDataRec135 : STRUCT
         majMinVer  : Byte := BYTE#0;   // Major / minor version
         dataRecordNum  : Byte := BYTE#151;   // Data record number for data record mapping = 151
         numMeasValues  : Byte := BYTE#150;   // Number of measured values for data record mapping
         resb3  : Byte;   // Reserved
         measValueID  : Array[1..150] of Word;   // ID of measured value for data record mapping
      END_STRUCT;

   END_TYPE

   TYPE EMHFDataRec151Real : STRUCT
         version  : Byte;   // Version
         numMeasValues  : Byte := BYTE#150;   // Number of measured values
         measValue  : Array[1..150] of Real;   // ID of measured value
      END_STRUCT;

   END_TYPE

   TYPE MotorStarterOut : STRUCT
         motorCw : Bool;   // Motor CW
         motorCcw : Bool;   // Motor CCW (Reversing starters only)
         res02 : Bool;   // Reserved
         tripReset : Bool;   // Trip RESET
         emergencyStart : Bool;   // Emergency start
         res05 : Bool;   // Reserved
         res06 : Bool;   // Reserved
         coldStart : Bool;   // Cold start
         res10 : Bool;   // Reserved
         res11 : Bool;   // Reserved
         res12 : Bool;   // Reserved
         res13 : Bool;   // Reserved
         res14 : Bool;   // Reserved
         res15 : Bool;   // Reserved
         res16 : Bool;   // Reserved
         disableQuickStop : Bool;   // Disable quick stop
      END_STRUCT;

   END_TYPE

   TYPE TMPulseControlFrequ : STRUCT
         channel : Array[0..1] of TMPulseControlFrequCh;
      END_STRUCT;

   END_TYPE

   TYPE EEatIndustryProfileE2 : STRUCT
         totalActivePower  : Real;   // Total active power L1 L2 L3
         totalActiveEnergyIn  : Real;   // Total active energy inflow L1 L2 L3
         totalActiveEnergyOut  : Real;   // Total active energy outflow L1 L2 L3
      END_STRUCT;

   END_TYPE

   TYPE EEatIndustryProfileE3 : STRUCT
         activePowerL1  : Real;   // Active power L1
         activePowerL2  : Real;   // Active power L2
         activePowerL3  : Real;   // Active power L3
         reactivePowerQtotL1  : Real;   // Reactive power Qtot L1
         reactivePowerQtotL2  : Real;   // Reactive power Qtot L2
         reactivePowerQtotL3  : Real;   // Reactive power Qtot L2
         totalActiveEnergyInLong  : LReal;   // Total active energy inflow L1 L2 L3
         totalActiveEnergyOutLong  : LReal;   // Total active energy outflow L1 L2 L3
         totalReactiveEnergyInLong  : LReal;   // Total reactive energy inflow L1 L2 L3
         totalReactiveEnergyOutLong  : LReal;   // Total reactive energy outflow L1 L2 L3
         voltL1N  : Real;   // Voltage UL1-N
         voltL2N  : Real;   // Voltage UL2-N
         voltL3N  : Real;   // Voltage UL3-N
         voltL1L2  : Real;   // Voltage UL1-L2
         voltL2L3  : Real;   // Voltage UL2-L3
         voltL3L1  : Real;   // Voltage UL3-L1
         currentL1  : Real;   // Current L1
         currentL2  : Real;   // Current L2
         currentL3  : Real;   // Current L3
         powerFactorL1  : Real;   // Power factor L1
         powerFactorL2  : Real;   // Power factor L2
         powerFactorL3  : Real;   // Power factor L3
      END_STRUCT;

   END_TYPE

   TYPE EM480VSTDataRec145 : STRUCT
         version  : Byte;   // Version
         resb1  : Byte;   // Reserved
         minVoltL1N  : Real;   // Min. voltage UL1-N
         minVoltL2N  : Real;   // Min. voltage UL2-N
         minVoltL3N  : Real;   // Min. voltage UL3-N
         minVoltL1L2  : Real;   // Min. voltage UL1-L2
         minVoltL2L3  : Real;   // Min. voltage UL2-L3
         minVoltL3L1  : Real;   // Min. voltage UL3-L1
         minCurrentL1  : Real;   // Min. current L1
         minCurrentL2  : Real;   // Min. current L2
         minCurrentL3  : Real;   // Min. current L3
         minApparentPowerL1  : Real;   // Min. apparent power L1
         minApparentPowerL2  : Real;   // Min. apparent power L2
         minApparentPowerL3  : Real;   // Min. apparent power L3
         minActivePowerL1  : Real;   // Min. active power L1
         minActivePowerL2  : Real;   // Min. active power L2
         minActivePowerL3  : Real;   // Min. active power L3
         minReactivePowerL1  : Real;   // Min. reactive power L1
         minReactivePowerL2  : Real;   // Min. reactive power L2
         minReactivePowerL3  : Real;   // Min. reactive power L3
         minPowerFactorL1  : Real;   // Min. power factor L1
         minPowerFactorL2  : Real;   // Min. power factor L2
         minPowerFactorL3  : Real;   // Min. power factor L3
         minFrequency  : Real;   // Min. frequency
         minTotalApparentPower  : Real;   // Min. total apparent power
         minTotalActivePower  : Real;   // Min. total active power
         minTotalReactivePower  : Real;   // Min. total reactive power
         minTotalPowerFactor  : Real;   // Min. total power factor
      END_STRUCT;

   END_TYPE

   TYPE EM480VHFDataRec144V1 : STRUCT
         version  : Byte;   // Version
         resb1  : Byte;   // Reserved
         maxVoltL1N  : Real;   // Max. voltage UL1-N
         maxVoltL2N  : Real;   // Max. voltage UL2-N
         maxVoltL3N  : Real;   // Max. voltage UL3-N
         maxVoltL1L2  : Real;   // Max. voltage UL1-L2
         maxVoltL2L3  : Real;   // Max. voltage UL2-L3
         maxVoltL3L1  : Real;   // Max. voltage UL3-L1
         maxCurrentL1  : Real;   // Max. current L1
         maxCurrentL2  : Real;   // Max. current L2
         maxCurrentL3  : Real;   // Max. current L3
         maxApparentPowerL1  : Real;   // Max. apparent power L1
         maxApparentPowerL2  : Real;   // Max. apparent power L2
         maxApparentPowerL3  : Real;   // Max. apparent power L3
         maxActivePowerL1  : Real;   // Max. active power L1
         maxActivePowerL2  : Real;   // Max. active power L2
         maxActivePowerL3  : Real;   // Max. active power L3
         maxReactivePowerQtotL1  : Real;   // Max. reactive power Qtot L1
         maxReactivePowerQtotL2  : Real;   // Max. reactive power Qtot L2
         maxReactivePowerQtotL3  : Real;   // Max. reactive power Qtot L3
         maxPowerFactorL1  : Real;   // Max. power factor L1
         maxPowerFactorL2  : Real;   // Max. power factor L2
         maxPowerFactorL3  : Real;   // Max. power factor L3
         maxFrequency  : Real;   // Max. frequency
         maxTotalApparentPower  : Real;   // Max. apparent power L1 L2 L3
         maxTotalActivePower  : Real;   // Max. active power L1 L2 L3
         maxTotalReactivePowerQtot  : Real;   // Max. reactive power Qtot L1 L2 L3
         maxTotalPowerFactor  : Real;   // Max. power factor λ L1L2L3
         maxReactivePowerQnL1  : Real;   // Max. reactive power Qn L1
         maxReactivePowerQnL2  : Real;   // Max. reactive power Qn L2
         maxReactivePowerQnL3  : Real;   // Max. reactive power Qn L3
         maxMeanVoltLN  : Real;   // Max. mean voltage L-N
         maxMeanVoltLL  : Real;   // Max. mean voltage L-L
         maxSumMeanCurr  : Real;   // Max. sum mean value current
         maxFundVoltL1  : Real;   // Max. fundamental voltage L1
         maxFundVoltL2  : Real;   // Max. fundamental voltage L2
         maxFundVoltL3  : Real;   // Max. fundamental voltage L3
         maxFundCurrL1  : Real;   // Max. fundamental current L1
         maxFundCurrL2  : Real;   // Max. fundamental current L2
         maxFundCurrL3  : Real;   // Max. fundamental current L3
         maxFundApparentPowerL1  : Real;   // Max. fundamental apparent power L1
         maxFundApparentPowerL2  : Real;   // Max. fundamental apparent power L2
         maxFundApparentPowerL3  : Real;   // Max. fundamental apparent power L3
         maxFundReactivePowerL1  : Real;   // Max. fundamental reactive power L1
         maxFundReactivePowerL2  : Real;   // Max. fundamental reactive power L2
         maxFundReactivePowerL3  : Real;   // Max. fundamental reactive power L3
         maxFundActivePowerL1  : Real;   // Max. fundamental active power L1
         maxFundActivePowerL2  : Real;   // Max. fundamental active power L2
         maxFundActivePowerL3  : Real;   // Max. fundamental active power L3
         maxFundActiveFactorL1  : Real;   // Max. fundamental cos φ active factor L1
         maxFundActiveFactorL2  : Real;   // Max. fundamental cos φ active factor L2
         maxFundActiveFactorL3  : Real;   // Max. fundamental cos φ active factor L3
         maxTHDaNVoltL1  : Real;   // Max. THD+N voltage L1
         maxTHDaNVoltL2  : Real;   // Max. THD+N voltage L2
         maxTHDaNVoltL3  : Real;   // Max. THD+N voltage L3
         maxTHDaNCurrL1  : Real;   // Max. THD+N current L1
         maxTHDaNCurrL2  : Real;   // Max. THD+N current L2
         maxTHDaNCurrL3  : Real;   // Max. THD+N current L3
      END_STRUCT;

   END_TYPE

   TYPE EM480VSTDataRec144 : STRUCT
         version  : Byte;   // Version
         resb1  : Byte;   // Reserved
         maxVoltL1N  : Real;   // Max. voltage UL1-N
         maxVoltL2N  : Real;   // Max. voltage UL2-N
         maxVoltL3N  : Real;   // Max. voltage UL3-N
         maxVoltL1L2  : Real;   // Max. voltage UL1-L2
         maxVoltL2L3  : Real;   // Max. voltage UL2-L3
         maxVoltL3L1  : Real;   // Max. voltage UL3-L1
         maxCurrentL1  : Real;   // Max. current L1
         maxCurrentL2  : Real;   // Max. current L2
         maxCurrentL3  : Real;   // Max. current L3
         maxApparentPowerL1  : Real;   // Max. apparent power L1
         maxApparentPowerL2  : Real;   // Max. apparent power L2
         maxApparentPowerL3  : Real;   // Max. apparent power L3
         maxActivePowerL1  : Real;   // Max. active power L1
         maxActivePowerL2  : Real;   // Max. active power L2
         maxActivePowerL3  : Real;   // Max. active power L3
         maxReactivePowerL1  : Real;   // Max. reactive power L1
         maxReactivePowerL2  : Real;   // Max. reactive power L2
         maxReactivePowerL3  : Real;   // Max. reactive power L3
         maxPowerFactorL1  : Real;   // Max. power factor L1
         maxPowerFactorL2  : Real;   // Max. power factor L2
         maxPowerFactorL3  : Real;   // Max. power factor L3
         maxFrequency  : Real;   // Max. frequency
         maxTotalApparentPower  : Real;   // Max. total apparent power
         maxTotalActivePower  : Real;   // Max. total active power
         maxTotalReactivePower  : Real;   // Max. total reactive power
         maxTotalPowerFactor  : Real;   // Max. total power factor
      END_STRUCT;

   END_TYPE

   TYPE EM480VSTDataRec143 : STRUCT
         version  : Byte := BYTE#1;   // Version
         resb1  : Byte;   // Reserved
         controlStatusByte1L1  : Byte;   // Status / control byte 1 - L1
         controlStatusByte2L1  : Byte;   // Status / control byte 2 - L1
         controlStatusByte1L2  : Byte;   // Status / control byte 1 - L2
         controlStatusByte2L2  : Byte;   // Status / control byte 2 - L2
         controlStatusByte1L3  : Byte;   // Status / control byte 1 - L3
         controlStatusByte2L3  : Byte;   // Status / control byte 2 - L3
         activeEnergyInL1  : LReal;   // Active energy inflow (initial value) L1
         activeEnergyOutL1  : LReal;   // Active energy outflow (initial value) L1
         reactiveEnergyInL1  : LReal;   // Reactive energy inflow (initial value) L1
         reactiveEnergyOutL1  : LReal;   // Reactive energy outflow (initial value) L1
         apparentEnergyL1  : LReal;   // Apparent energy (initial value) L1
         activeEnergyInL2  : LReal;   // Active energy inflow (initial value) L2
         activeEnergyOutL2  : LReal;   // Active energy outflow (initial value) L2
         reactiveEnergyInL2  : LReal;   // Reactive energy inflow (initial value) L2
         reactiveEnergyOutL2  : LReal;   // Reactive energy outflow (initial value) L2
         apparentEnergyL2  : LReal;   // Apparent energy (initial value) L2
         activeEnergyInL3  : LReal;   // Active energy inflow (initial value) L3
         activeEnergyOutL3  : LReal;   // Active energy outflow (initial value) L3
         reactiveEnergyInL3  : LReal;   // Reactive energy inflow (initial value) L3
         reactiveEnergyOutL3  : LReal;   // Reactive energy outflow (initial value) L3
         apparentEnergyL3  : LReal;   // Apparent energy (initial value) L3
         ovCntActiveEnergyInL1  : UInt;   // Overflow counter active energy inflow L1
         ovCntActiveEnergyOutL1  : UInt;   // Overflow counter active energy outflow L1
         ovCntReactiveEnergyInL1  : UInt;   // Overflow counter reactive energy inflow L1
         ovCntReactiveEnergyOutL1  : UInt;   // Overflow counter reactive energy outflow L1
         ovCntApparentEnergyL1  : UInt;   // Overflow counter apparent energy L1
         ovCntActiveEnergyInL2  : UInt;   // Overflow counter active energy inflow L2
         ovCntActiveEnergyOutL2  : UInt;   // Overflow counter active energy outflow L2
         ovCntReactiveEnergyInL2  : UInt;   // Overflow counter reactive energy inflow L2
         ovCntReactiveEnergyOutL2  : UInt;   // Overflow counter reactive energy outflow L2
         ovCntApparentEnergyL2  : UInt;   // Overflow counter apparent energy L2
         ovCntActiveEnergyInL3  : UInt;   // Overflow counter active energy inflow L3
         ovCntActiveEnergyOutL3  : UInt;   // Overflow counter active energy outflow L3
         ovCntReactiveEnergyInL3  : UInt;   // Overflow counter reactive energy inflow L3
         ovCntReactiveEnergyOutL3  : UInt;   // Overflow counter reactive energy outflow L3
         ovCntApparentEnergyL3  : UInt;   // Overflow counter apparent energy L3
         operHoursCntL1  : Real;   // Operating hours counter L1 (initial value)
         operHoursCntL2  : Real;   // Operating hours counter L2 (initial value)
         operHoursCntL3  : Real;   // Operating hours counter L2 (initial value)
      END_STRUCT;

   END_TYPE

   TYPE EM480VSTDataRec142 : STRUCT
         version  : Byte := BYTE#1;   // Version
         resb1  : Byte;   // Reserved
         voltL1N  : Real;   // Voltage UL1-N
         voltL2N  : Real;   // Voltage UL2-N
         voltL3N  : Real;   // Voltage UL3-N
         voltL1L2  : Real;   // Voltage UL1-L2
         voltL2L3  : Real;   // Voltage UL2-L3
         voltL3L1  : Real;   // Voltage UL3-L1
         currentL1  : Real;   // Current L1
         currentL2  : Real;   // Current L2
         currentL3  : Real;   // Current L3
         powerFactorL1  : Real;   // Power factor L1
         powerFactorL2  : Real;   // Power factor L2
         powerFactorL3  : Real;   // Power factor L3
         totalPowerFactor  : Real;   // Total power factor L1 L2 L3
         frequency  : Real;   // Frequency
         amplUnbalanceVolt  : Real;   // Amplitude unbalance for voltage
         amplUnbalanceCurrent  : Real;   // Amplitude unbalance for current
         apparentPowerL1  : Real;   // Apparent power L1
         apparentPowerL2  : Real;   // Apparent power L2
         apparentPowerL3  : Real;   // Apparent power L3
         totalApparentPower  : Real;   // Total apparent power L1 L2 L3
         reactivePowerL1  : Real;   // Reactive power L1
         reactivePowerL2  : Real;   // Reactive power L2
         reactivePowerL3  : Real;   // Reactive power L2
         totalReactivePower  : Real;   // Total reactive power L1 L2 L3
         activePowerL1  : Real;   // Active power L1
         activePowerL2  : Real;   // Active power L2
         activePowerL3  : Real;   // Active power L3
         totalActivePower  : Real;   // Total active power L1 L2 L3
         phaseAngleL1  : Real;   //  Phase angle L1
         phaseAngleL2  : Real;   //  Phase angle L2
         phaseAngleL3  : Real;   //  Phase angle L3
         totalApparentEnergy  : Real;   // Total apparent energy L1 L2 L3
         totalReactiveEnergy  : Real;   // Total reactive energy L1 L2 L3
         totalActiveEnergy  : Real;   // Total active energy L1 L2 L3
         totalReactiveEnergyIn  : Real;   // Total reactive energy inflow L1 L2 L3
         totalReactiveEnergyOut  : Real;   // Total reactive energy outflow L1 L2 L3
         totalActiveEnergyIn  : Real;   // Total active energy inflow L1 L2 L3
         totalActiveEnergyOut  : Real;   // Total active energy outflow L1 L2 L3
         totalApparentEnergyLong  : LReal;   // Total apparent energy L1 L2 L3
         totalReactiveEnergyLong  : LReal;   // Total reactive energy L1 L2 L3
         totalActiveEnergyLong  : LReal;   // Total active energy L1 L2 L3
         totalReactiveEnergyInLong  : LReal;   // Total reactive energy inflow L1 L2 L3
         totalReactiveEnergyOutLong  : LReal;   // Total reactive energy outflow L1 L2 L3
         totalActiveEnergyInLong  : LReal;   // Total active energy inflow L1 L2 L3
         totalActiveEnergyOutLong  : LReal;   // Total active energy outflow L1 L2 L3
         neutralCurrent  : Real;   // Neutral current
      END_STRUCT;

   END_TYPE

   TYPE EM480VHFDataRec142V3 : STRUCT
         version  : Byte := BYTE#3;   // Version
         resb1  : Byte;   // Reserved
         voltL1N  : Real;   // Voltage UL1-N
         voltL2N  : Real;   // Voltage UL2-N
         voltL3N  : Real;   // Voltage UL3-N
         voltL1L2  : Real;   // Voltage UL1-L2
         voltL2L3  : Real;   // Voltage UL2-L3
         voltL3L1  : Real;   // Voltage UL3-L1
         currentL1  : Real;   // Current L1
         currentL2  : Real;   // Current L2
         currentL3  : Real;   // Current L3
         powerFactorL1  : Real;   // Power factor L1
         powerFactorL2  : Real;   // Power factor L2
         powerFactorL3  : Real;   // Power factor L3
         totalPowerFactor  : Real;   // Total power factor L1 L2 L3
         frequency  : Real;   // Frequency
         amplUnbalanceVolt  : Real;   // Amplitude unbalance for voltage
         amplUnbalanceCurrent  : Real;   // Amplitude unbalance for current
         apparentPowerL1  : Real;   // Apparent power L1
         apparentPowerL2  : Real;   // Apparent power L2
         apparentPowerL3  : Real;   // Apparent power L3
         totalApparentPower  : Real;   // Total apparent power L1 L2 L3
         reactivePowerQtotL1  : Real;   // Reactive power Qtot L1
         reactivePowerQtotL2  : Real;   // Reactive power Qtot L2
         reactivePowerQtotL3  : Real;   // Reactive power Qtot L2
         totalReactivePowerQtot  : Real;   // Total reactive power Qtot L1 L2 L3
         activePowerL1  : Real;   // Active power L1
         activePowerL2  : Real;   // Active power L2
         activePowerL3  : Real;   // Active power L3
         totalActivePower  : Real;   // Total active power L1 L2 L3
         phaseAngleL1  : Real;   //  Phase angle L1
         phaseAngleL2  : Real;   //  Phase angle L2
         phaseAngleL3  : Real;   //  Phase angle L3
         totalApparentEnergy  : Real;   // Total apparent energy L1 L2 L3
         totalReactiveEnergy  : Real;   // Total reactive energy L1 L2 L3
         totalActiveEnergy  : Real;   // Total active energy L1 L2 L3
         totalReactiveEnergyIn  : Real;   // Total reactive energy inflow L1 L2 L3
         totalReactiveEnergyOut  : Real;   // Total reactive energy outflow L1 L2 L3
         totalActiveEnergyIn  : Real;   // Total active energy inflow L1 L2 L3
         totalActiveEnergyOut  : Real;   // Total active energy outflow L1 L2 L3
         totalApparentEnergyLong  : LReal;   // Total apparent energy L1 L2 L3
         totalReactiveEnergyLong  : LReal;   // Total reactive energy L1 L2 L3
         totalActiveEnergyLong  : LReal;   // Total active energy L1 L2 L3
         totalReactiveEnergyInLong  : LReal;   // Total reactive energy inflow L1 L2 L3
         totalReactiveEnergyOutLong  : LReal;   // Total reactive energy outflow L1 L2 L3
         totalActiveEnergyInLong  : LReal;   // Total active energy inflow L1 L2 L3
         totalActiveEnergyOutLong  : LReal;   // Total active energy outflow L1 L2 L3
         neutralCurrent  : Real;   // Neutral current
         neutralCurrentCyc10to12  : Real;   // Neutral current 10/12 cycle
         reactivePowerQnL1  : Real;   // Reactive power Qn L1
         reactivePowerQnL2  : Real;   // Reactive power Qn L2
         reactivePowerQnL3  : Real;   // Reactive power Qn L3
         totalReactivePowerQn  : Real;   // Total reactive power Qn L1 L2 L3
         averageVoltLN  : Real;   // Average voltage L-N (Usum)
         averageVoltLL  : Real;   // Average voltage L-L
         totalAverageCurr  : Real;   // Average current L1L2L3 (Isum)
         totalMeanPowerFactor  : Real;   // Mean power factor λ L1L2L3
         fundVoltL1  : Real;   // Fundamental voltage L1
         fundVoltL2  : Real;   // Fundamental voltage L2
         fundVoltL3  : Real;   // Fundamental voltage L3
         fundCurrL1  : Real;   // Fundamental current L1
         fundCurrL2  : Real;   // Fundamental current L2
         fundCurrL3  : Real;   // Fundamental current L3
         fundApparentPowerL1  : Real;   // Fundamental apparent power L1
         fundApparentPowerL2  : Real;   // Fundamental apparent power L2
         fundApparentPowerL3  : Real;   // Fundamental apparent power L3
         fundReactivePowerL1  : Real;   // Fundamental reactive power L1
         fundReactivePowerL2  : Real;   // Fundamental reactive power L2
         fundReactivePowerL3  : Real;   // Fundamental reactive power L3
         fundActivePowerL1  : Real;   // Fundamental active power L1
         fundActivePowerL2  : Real;   // Fundamental active power L2
         fundActivePowerL3  : Real;   // Fundamental active power L3
         fundActiveFactorL1  : Real;   // Fundamental cos φ active factor L1
         fundActiveFactorL2  : Real;   // Fundamental cos φ active factor L2
         fundActiveFactorL3  : Real;   // Fundamental cos φ active factor L3
         harmDistTHDaNVoltL1  : Real;   // Harmonic distortion (THD+N) voltage L1
         harmDistTHDaNVoltL2  : Real;   // Harmonic distortion (THD+N) voltage L2
         harmDistTHDaNVoltL3  : Real;   // Harmonic distortion (THD+N) voltage L3
         harmDistTHDaNCurrL1  : Real;   // Harmonic distortion (THD+N) current L1
         harmDistTHDaNCurrL2  : Real;   // Harmonic distortion (THD+N) current L2
         harmDistTHDaNCurrL3  : Real;   // Harmonic distortion (THD+N) current L3
         currentModuleTime  : PNIOTimeStamp;   // Current module time
      END_STRUCT;

   END_TYPE

   TYPE EM400VSTDataRec143 : STRUCT
         version  : Byte;   // Version
         resb1  : Byte;   // Reserved
         controlByte1L1  : Byte;   // Control byte 1 - L1
         controlByte2L1  : Byte;   // Control byte 2 - L1
         controlByte1L2  : Byte;   // Control byte 1 - L2
         controlByte2L2  : Byte;   // Control byte 2 - L2
         controlByte1L3  : Byte;   // Control byte 1 - L3
         controlByte2L3  : Byte;   // Control byte 2 - L3
         activeEnergyInL1  : LReal;   // Active energy inflow (initial value) L1
         activeEnergyOutL1  : LReal;   // Active energy outflow (initial value) L1
         reactiveEnergyInL1  : LReal;   // Reactive energy inflow (initial value) L1
         reactiveEnergyOutL1  : LReal;   // Reactive energy outflow (initial value) L1
         apparentEnergyL1  : LReal;   // Apparent energy (initial value) L1
         activeEnergyInL2  : LReal;   // Active energy inflow (initial value) L2
         activeEnergyOutL2  : LReal;   // Active energy outflow (initial value) L2
         reactiveEnergyInL2  : LReal;   // Reactive energy inflow (initial value) L2
         reactiveEnergyOutL2  : LReal;   // Reactive energy outflow (initial value) L2
         apparentEnergyL2  : LReal;   // Apparent energy (initial value) L2
         activeEnergyInL3  : LReal;   // Active energy inflow (initial value) L3
         activeEnergyOutL3  : LReal;   // Active energy outflow (initial value) L3
         reactiveEnergyInL3  : LReal;   // Reactive energy inflow (initial value) L3
         reactiveEnergyOutL3  : LReal;   // Reactive energy outflow (initial value) L3
         apparentEnergyL3  : LReal;   // Apparent energy (initial value) L3
      END_STRUCT;

   END_TYPE

   TYPE EM480VSTDataRec150 : STRUCT
         version  : Byte := BYTE#1;   // Version
         resb1  : Byte;   // Reserved
         operHoursCntTotal  : Real;   // Operating hours counter L1 L2 L3
         operHoursCntL1  : Real;   // Operating hours counter L1
         operHoursCntL2  : Real;   // Operating hours counter L2
         operHoursCntL3  : Real;   // Operating hours counter L3
         statusLimViolGW1to16  : Word;   // Status limit violation GW 1...16
         statusEnergyCntOv  : Word;   // Status of energy counter overflows
         cntLimViolGw1  : UDInt;   // Counter limit violation GW 1
         cntLimViolGw2  : UDInt;   // Counter limit violation GW 2
         cntLimViolGw3  : UDInt;   // Counter limit violation GW 3
         cntLimViolGw4  : UDInt;   // Counter limit violation GW 4
         cntLimViolGw5  : UDInt;   // Counter limit violation GW 5
         cntLimViolGw6  : UDInt;   // Counter limit violation GW 6
         cntLimViolGw7  : UDInt;   // Counter limit violation GW 7
         cntLimViolGw8  : UDInt;   // Counter limit violation GW 8
         cntLimViolGw9  : UDInt;   // Counter limit violation GW 9
         cntLimViolGw10  : UDInt;   // Counter limit violation GW 10
         cntLimViolGw11  : UDInt;   // Counter limit violation GW 11
         cntLimViolGw12  : UDInt;   // Counter limit violation GW 12
         cntLimViolGw13  : UDInt;   // Counter limit violation GW 13
         cntLimViolGw14  : UDInt;   // Counter limit violation GW 14
         cntLimViolGw15  : UDInt;   // Counter limit violation GW 15
         cntLimViolGw16  : UDInt;   // Counter limit violation GW 16
         qualifierL1L2L3  : Word;   // Qualifier L1 L2 L3
      END_STRUCT;

   END_TYPE

   TYPE EM480VSTDataRec149 : STRUCT
         version  : Byte := BYTE#1;   // Version
         resb1  : Byte;   // Reserved
         qualifierL3  : Word;   // Qualifier L3
         voltL3N  : Real;   // Voltage UL3-N
         currentL3  : Real;   // Current L3
         apparentPowerL3  : Real;   // Apparent power L3
         activePowerL3  : Real;   // Active power L3
         reactivePowerL3  : Real;   // Reactive power L3
         powerFactorL3  : Real;   // Power factor L3
         phaseAngleL3  : Real;   // Phase angle L3
         apparentEnergyL3  : LReal;   // Apparent energy L3
         activeEnergyL3  : LReal;   // Active energy (total) L3
         reactiveEnergyL3  : LReal;   // Reactive energy (total) L3
         maxVoltL3N  : Real;   // Max. voltage UL3-N
         maxCurrentL3  : Real;   // Max. current L3
         maxApparentPowerL3  : Real;   // Max. apparent power L3
         maxActivePowerL3  : Real;   // Max. active power L3
         maxReactivePowerL3  : Real;   // Max. reactive power L3
         maxPowerFactorL3  : Real;   // Max. power factor L3
         minVoltL3N  : Real;   // Min. voltage UL3-N
         minCurrentL3  : Real;   // Min. current L3
         minApparentPowerL3  : Real;   // Min. apparent power L3
         minActivePowerL3  : Real;   // Min. active power L3
         minReactivePowerL3  : Real;   // Min. reactive power L3
         minPowerFactorL3  : Real;   // Min. power factor L3
      END_STRUCT;

   END_TYPE

   TYPE EM480VSTDataRec148 : STRUCT
         version  : Byte := BYTE#1;   // Version
         resb1  : Byte;   // Reserved
         qualifierL2  : Word;   // Qualifier L2
         voltL2N  : Real;   // Voltage UL2-N
         currentL2  : Real;   // Current L2
         apparentPowerL2  : Real;   // Apparent power L2
         activePowerL2  : Real;   // Active power L2
         reactivePowerL2  : Real;   // Reactive power L2
         powerFactorL2  : Real;   // Power factor L2
         phaseAngleL2  : Real;   // Phase angle L2
         apparentEnergyL2  : LReal;   // Apparent energy L2
         activeEnergyL2  : LReal;   // Active energy (total) L2
         reactiveEnergyL2  : LReal;   // Reactive energy (total) L2
         maxVoltL2N  : Real;   // Max. voltage UL2-N
         maxCurrentL2  : Real;   // Max. current L2
         maxApparentPowerL2  : Real;   // Max. apparent power L2
         maxActivePowerL2  : Real;   // Max. active power L2
         maxReactivePowerL2  : Real;   // Max. reactive power L2
         maxPowerFactorL2  : Real;   // Max. power factor L2
         minVoltL2N  : Real;   // Min. voltage UL2-N
         minCurrentL2  : Real;   // Min. current L2
         minApparentPowerL2  : Real;   // Min. apparent power L2
         minActivePowerL2  : Real;   // Min. active power L2
         minReactivePowerL2  : Real;   // Min. reactive power L2
         minPowerFactorL2  : Real;   // Min. power factor L2
      END_STRUCT;

   END_TYPE

   TYPE EM480VSTDataRec147 : STRUCT
         version  : Byte := BYTE#1;   // Version
         resb1  : Byte;   // Reserved
         qualifierL1  : Word;   // Qualifier L1
         voltL1N  : Real;   // Voltage UL1-N
         currentL1  : Real;   // Current L1
         apparentPowerL1  : Real;   // Apparent power L1
         activePowerL1  : Real;   // Active power L1
         reactivePowerL1  : Real;   // Reactive power L1
         powerFactorL1  : Real;   // Power factor L1
         phaseAngleL1  : Real;   // Phase angle L1
         apparentEnergyL1  : LReal;   // Apparent energy L1
         totalActiveEnergyL1  : LReal;   // Active energy (total) L1
         totalReactiveEnergyL1  : LReal;   // Reactive energy (total) L1
         maxVoltL1N  : Real;   // Max. voltage UL1-N
         maxCurrentL1  : Real;   // Max. current L1
         maxApparentPowerL1  : Real;   // Max. apparent power L1
         maxActivePowerL1  : Real;   // Max. active power L1
         maxReactivePowerL1  : Real;   // Max. reactive power L1
         maxPowerFactorL1  : Real;   // Max. power factor L1
         minVoltL1N  : Real;   // Min. voltage UL1-N
         minCurrentL1  : Real;   // Min. current L1
         minApparentPowerL1  : Real;   // Min. apparent power L1
         minActivePowerL1  : Real;   // Min. active power L1
         minReactivePowerL1  : Real;   // Min. reactive power L1
         minPowerFactorL1  : Real;   // Min. power factor L1
      END_STRUCT;

   END_TYPE

   TYPE EM480VHFDataRec170 : STRUCT
         version  : Byte;   // Version
         resb1  : Byte;   // Reserved
         numIDs  : UInt;   // Number of IDs
         measValueID  : Array[1..580] of UInt;   // ID measured value
      END_STRUCT;

   END_TYPE

   TYPE EM400VSTDataRec128 : STRUCT
         majMinVer  : Byte := BYTE#65;   // Major / minor version
         numParamStruct  : Byte := BYTE#2;   // Number of parameter structures = 2
         numModuleParamBlocks  : Byte := BYTE#1;   // Number of module parameter blocks = 1
         lengthModuleParamBlock  : Byte := BYTE#8;   // Length of module parameter block = 8
         connectTypePhases  : Byte := BYTE#0;   // Connection type of the phases
         measRangePower  : Byte;   // Voltage measuring range of the power supply system
         energyCountGateLineFrequ  : Byte;   // Energy counter gate / Line frequency of the power supply system
         lineVoltTolerance  : Byte;   // Line voltage tolerance
         diagLineVolt  : Byte;   // Diagnostics line voltage
         lowLimitCurrMeas  : Byte;   // Low limit for current measurement [mA]
         resb10  : Byte;   // Reserved
         idUserDataVariant  : Byte;   // ID of the user data variant
         numChannelParamBlocks  : Byte := BYTE#3;   // Number of channel parameter blocks = 3
         lengthChannelParamBlock  : Byte := BYTE#8;   // Length of channel parameter block = 8
         channel  : Array[0..2] of EMSTDataRecCh;
      END_STRUCT;

   END_TYPE

   TYPE EEatIndustryProfileE1 : STRUCT
         totalActivePower  : Real;   // Total active power L1 L2 L3
      END_STRUCT;

   END_TYPE

   TYPE EMSTDataRec128 : STRUCT
         majMinVer  : Byte := BYTE#64;   // Major / minor version
         numParamStruct  : Byte := BYTE#2;   // Number of parameter structures = 2
         numModuleParamBlocks  : Byte := BYTE#1;   // Number of module parameter blocks = 1
         lengthModuleParamBlock  : Byte := BYTE#8;   // Length of module parameter block = 8
         connectTypePhases  : Byte := BYTE#0;   // Connection type of the phases
         measRangePower  : Byte;   // Voltage measuring range of the power supply system
         energyCountGateLineFrequ  : Byte;   // Energy counter gate / Line frequency of the power supply system
         lineVoltTolerance  : Byte;   // Line voltage tolerance
         diagLineVolt  : Byte;   // Diagnostics line voltage
         lowLimitCurrMeas  : Byte;   // Low limit for current measurement [mA]
         resb10  : Byte;   // Reserved
         idUserDataVariant  : Byte;   // ID of the user data variant
         numChannelParamBlocks  : Byte := BYTE#3;   // Number of channel parameter blocks = 3
         lengthChannelParamBlock  : Byte := BYTE#8;   // Length of channel parameter block = 8
         channel  : Array[0..2] of EMSTDataRecCh;
      END_STRUCT;

   END_TYPE

   TYPE EEatIndustryProfileE0 : STRUCT
         currentL1  : Real;   // Current L1
         currentL2  : Real;   // Current L2
         currentL3  : Real;   // Current L3
      END_STRUCT;

   END_TYPE

   TYPE EM480VHFDataRec147V0 : STRUCT
         version  : Byte;   // Version
         resb1  : Byte;   // Reserved
         qualifierL1  : Word;   // Qualifier L1
         voltL1N  : Real;   // Voltage UL1-N
         currentL1  : Real;   // Current L1
         apparentPowerL1  : Real;   // Apparent power L1
         activePowerL1  : Real;   // Active power L1
         reactivePowerQtotL1  : Real;   // Reactive power Qtot L1
         powerFactorL1  : Real;   // Power factor L1
         phaseAngleL1  : Real;   // Phase angle L1
         apparentEnergyLongL1  : LReal;   // Apparent energy L1
         totalActiveEnergyLongL1  : LReal;   // Active energy (total) L1
         totalReactiveEnergyLongL1  : LReal;   // Reactive energy (total) L1
         maxVoltL1N  : Real;   // Max. voltage UL1-N
         maxCurrentL1  : Real;   // Max. current L1
         maxApparentPowerL1  : Real;   // Max. apparent power L1
         maxActivePowerL1  : Real;   // Max. active power L1
         maxReactivePowerQtotL1  : Real;   // Max. reactive power Qtot L1
         maxPowerFactorL1  : Real;   // Max. power factor L1
         minVoltL1N  : Real;   // Min. voltage UL1-N
         minCurrentL1  : Real;   // Min. current L1
         minApparentPowerL1  : Real;   // Min. apparent power L1
         minActivePowerL1  : Real;   // Min. active power L1
         minReactivePowerQtotL1  : Real;   // Min. reactive power Qtot L1
         minPowerFactorL1  : Real;   // Min. power factor L1
      END_STRUCT;

   END_TYPE

   TYPE EM480VHFDataRec155 : STRUCT
         version  : Byte := BYTE#1;   // Version
         resb1  : Byte;   // Reserved
         minVoltL1N  : RealValueAndPNIOTimeStamp;   // Min. voltage UL1-N
         minVoltL2N  : RealValueAndPNIOTimeStamp;   // Min. voltage UL2-N
         minVoltL3N  : RealValueAndPNIOTimeStamp;   // Min. voltage UL3-N
         minVoltL1L2  : RealValueAndPNIOTimeStamp;   // Min. voltage UL1-L2
         minVoltL2L3  : RealValueAndPNIOTimeStamp;   // Min. voltage UL2-L3
         minVoltL3L1  : RealValueAndPNIOTimeStamp;   // Min. voltage UL3-L1
         minCurrentL1  : RealValueAndPNIOTimeStamp;   // Min. current L1
         minCurrentL2  : RealValueAndPNIOTimeStamp;   // Min. current L2
         minCurrentL3  : RealValueAndPNIOTimeStamp;   // Min. current L3
         minApparentPowerL1  : RealValueAndPNIOTimeStamp;   // Min. apparent power L1
         minApparentPowerL2  : RealValueAndPNIOTimeStamp;   // Min. apparent power L2
         minApparentPowerL3  : RealValueAndPNIOTimeStamp;   // Min. apparent power L3
         minActivePowerL1  : RealValueAndPNIOTimeStamp;   // Min. active power L1
         minActivePowerL2  : RealValueAndPNIOTimeStamp;   // Min. active power L2
         minActivePowerL3  : RealValueAndPNIOTimeStamp;   // Min. active power L3
         minReactivePowerQtotL1  : RealValueAndPNIOTimeStamp;   // Min. reactive power Qtot L1
         minReactivePowerQtotL2  : RealValueAndPNIOTimeStamp;   // Min. reactive power Qtot L2
         minReactivePowerQtotL3  : RealValueAndPNIOTimeStamp;   // Min. reactive power Qtot L3
         minPowerFactorL1  : RealValueAndPNIOTimeStamp;   // Min. power factor L1
         minPowerFactorL2  : RealValueAndPNIOTimeStamp;   // Min. power factor L2
         minPowerFactorL3  : RealValueAndPNIOTimeStamp;   // Min. power factor L3
         minFrequency  : RealValueAndPNIOTimeStamp;   // Min. frequency
         minTotalApparentPower  : RealValueAndPNIOTimeStamp;   // Min. apparent power L1 L2 L3
         minTotalActivePower  : RealValueAndPNIOTimeStamp;   // Min. active power L1 L2 L3
         minTotalReactivePowerQn  : RealValueAndPNIOTimeStamp;   // Min. reactive power Qn L1 L2 L3
         minTotalPowerFactor  : RealValueAndPNIOTimeStamp;   // Min. power factor λ L1 L2 L3
         minReactivePowerQnL1  : RealValueAndPNIOTimeStamp;   // Min. reactive power Qn L1
         minReactivePowerQnL2  : RealValueAndPNIOTimeStamp;   // Min. reactive power Qn L2
         minReactivePowerQnL3  : RealValueAndPNIOTimeStamp;   // Min. reactive power Qn L3
         minMeanVoltLN  : RealValueAndPNIOTimeStamp;   // Min. mean voltage L-N
         minMeanVoltLL  : RealValueAndPNIOTimeStamp;   // Min. mean voltage L-L
         minTotalMeanCurr  : RealValueAndPNIOTimeStamp;   // Min. mean current L1 L2 L3
         minFundVoltL1  : RealValueAndPNIOTimeStamp;   // Min. fundamental voltage L1
         minFundVoltL2  : RealValueAndPNIOTimeStamp;   // Min. fundamental voltage L2
         minFundVoltL3  : RealValueAndPNIOTimeStamp;   // Min. fundamental voltage L3
         minFundCurrL1  : RealValueAndPNIOTimeStamp;   // Min. fundamental current L1
         minFundCurrL2  : RealValueAndPNIOTimeStamp;   // Min. fundamental current L2
         minFundCurrL3  : RealValueAndPNIOTimeStamp;   // Min. fundamental current L3
         minFundApparentPowerL1  : RealValueAndPNIOTimeStamp;   // Min. fundamental apparent power L1
         minFundApparentPowerL2  : RealValueAndPNIOTimeStamp;   // Min. fundamental apparent power L2
         minFundApparentPowerL3  : RealValueAndPNIOTimeStamp;   // Min. fundamental apparent power L3
         minFundReactivePowerL1  : RealValueAndPNIOTimeStamp;   // Min. fundamental reactive power L1
         minFundReactivePowerL2  : RealValueAndPNIOTimeStamp;   // Min. fundamental reactive power L2
         minFundReactivePowerL3  : RealValueAndPNIOTimeStamp;   // Min. fundamental reactive power L3
         minFundActivePowerL1  : RealValueAndPNIOTimeStamp;   // Min. fundamental active power L1
         minFundActivePowerL2  : RealValueAndPNIOTimeStamp;   // Min. fundamental active power L2
         minFundActivePowerL3  : RealValueAndPNIOTimeStamp;   // Min. fundamental active power L3
         minFundActiveFactorL1  : RealValueAndPNIOTimeStamp;   // Min. fundamental cos φ active factor L1
         minFundActiveFactorL2  : RealValueAndPNIOTimeStamp;   // Min. fundamental cos φ active factor L2
         minFundActiveFactorL3  : RealValueAndPNIOTimeStamp;   // Min. fundamental cos φ active factor L3
         minTHDaNVoltL1  : RealValueAndPNIOTimeStamp;   // Min. THD+N voltage L1
         minTHDaNVoltL2  : RealValueAndPNIOTimeStamp;   // Min. THD+N voltage L2
         minTHDaNVoltL3  : RealValueAndPNIOTimeStamp;   // Min. THD+N voltage L3
         minTHDaNCurrL1  : RealValueAndPNIOTimeStamp;   // Min. THD+N current L1
         minTHDaNCurrL2  : RealValueAndPNIOTimeStamp;   // Min. THD+N current L2
         minTHDaNCurrL3  : RealValueAndPNIOTimeStamp;   // Min. THD+N current L3
      END_STRUCT;

   END_TYPE

   TYPE EM480VHFDataRec154 : STRUCT
         version  : Byte := BYTE#1;   // Version
         resb1  : Byte;   // Reserved
         maxVoltL1N  : RealValueAndPNIOTimeStamp;   // Max. voltage UL1-N
         maxVoltL2N  : RealValueAndPNIOTimeStamp;   // Max. voltage UL2-N
         maxVoltL3N  : RealValueAndPNIOTimeStamp;   // Max. voltage UL3-N
         maxVoltL1L2  : RealValueAndPNIOTimeStamp;   // Max. voltage UL1-L2
         maxVoltL2L3  : RealValueAndPNIOTimeStamp;   // Max. voltage UL2-L3
         maxVoltL3L1  : RealValueAndPNIOTimeStamp;   // Max. voltage UL3-L1
         maxCurrentL1  : RealValueAndPNIOTimeStamp;   // Max. current L1
         maxCurrentL2  : RealValueAndPNIOTimeStamp;   // Max. current L2
         maxCurrentL3  : RealValueAndPNIOTimeStamp;   // Max. current L3
         maxApparentPowerL1  : RealValueAndPNIOTimeStamp;   // Max. apparent power L1
         maxApparentPowerL2  : RealValueAndPNIOTimeStamp;   // Max. apparent power L2
         maxApparentPowerL3  : RealValueAndPNIOTimeStamp;   // Max. apparent power L3
         maxActivePowerL1  : RealValueAndPNIOTimeStamp;   // Max. active power L1
         maxActivePowerL2  : RealValueAndPNIOTimeStamp;   // Max. active power L2
         maxActivePowerL3  : RealValueAndPNIOTimeStamp;   // Max. active power L3
         maxReactivePowerQtotL1  : RealValueAndPNIOTimeStamp;   // Max. reactive power Qtot L1
         maxReactivePowerQtotL2  : RealValueAndPNIOTimeStamp;   // Max. reactive power Qtot L2
         maxReactivePowerQtotL3  : RealValueAndPNIOTimeStamp;   // Max. reactive power Qtot L3
         maxPowerFactorL1  : RealValueAndPNIOTimeStamp;   // Max. power factor L1
         maxPowerFactorL2  : RealValueAndPNIOTimeStamp;   // Max. power factor L2
         maxPowerFactorL3  : RealValueAndPNIOTimeStamp;   // Max. power factor L3
         maxFrequency  : RealValueAndPNIOTimeStamp;   // Max. frequency
         maxTotalApparentPower  : RealValueAndPNIOTimeStamp;   // Max. apparent power L1 L2 L3
         maxTotalActivePower  : RealValueAndPNIOTimeStamp;   // Max. active power L1 L2 L3
         maxTotalReactivePowerQtot  : RealValueAndPNIOTimeStamp;   // Max. reactive power Qtot L1 L2 L3
         maxTotalPowerFactor  : RealValueAndPNIOTimeStamp;   // Max. power factor λ L1L2L3
         maxReactivePowerQnL1  : RealValueAndPNIOTimeStamp;   // Max. reactive power Qn L1
         maxReactivePowerQnL2  : RealValueAndPNIOTimeStamp;   // Max. reactive power Qn L2
         maxReactivePowerQnL3  : RealValueAndPNIOTimeStamp;   // Max. reactive power Qn L3
         maxMeanVoltLN  : RealValueAndPNIOTimeStamp;   // Max. mean voltage L-N
         maxMeanVoltLL  : RealValueAndPNIOTimeStamp;   // Max. mean voltage L-L
         maxSumMeanCurr  : RealValueAndPNIOTimeStamp;   // Max. sum mean value current
         maxFundVoltL1  : RealValueAndPNIOTimeStamp;   // Max. fundamental voltage L1
         maxFundVoltL2  : RealValueAndPNIOTimeStamp;   // Max. fundamental voltage L2
         maxFundVoltL3  : RealValueAndPNIOTimeStamp;   // Max. fundamental voltage L3
         maxFundCurrL1  : RealValueAndPNIOTimeStamp;   // Max. fundamental current L1
         maxFundCurrL2  : RealValueAndPNIOTimeStamp;   // Max. fundamental current L2
         maxFundCurrL3  : RealValueAndPNIOTimeStamp;   // Max. fundamental current L3
         maxFundApparentPowerL1  : RealValueAndPNIOTimeStamp;   // Max. fundamental apparent power L1
         maxFundApparentPowerL2  : RealValueAndPNIOTimeStamp;   // Max. fundamental apparent power L2
         maxFundApparentPowerL3  : RealValueAndPNIOTimeStamp;   // Max. fundamental apparent power L3
         maxFundReactivePowerL1  : RealValueAndPNIOTimeStamp;   // Max. fundamental reactive power L1
         maxFundReactivePowerL2  : RealValueAndPNIOTimeStamp;   // Max. fundamental reactive power L2
         maxFundReactivePowerL3  : RealValueAndPNIOTimeStamp;   // Max. fundamental reactive power L3
         maxFundActivePowerL1  : RealValueAndPNIOTimeStamp;   // Max. fundamental active power L1
         maxFundActivePowerL2  : RealValueAndPNIOTimeStamp;   // Max. fundamental active power L2
         maxFundActivePowerL3  : RealValueAndPNIOTimeStamp;   // Max. fundamental active power L3
         maxFundActiveFactorL1  : RealValueAndPNIOTimeStamp;   // Max. fundamental cos φ active factor L1
         maxFundActiveFactorL2  : RealValueAndPNIOTimeStamp;   // Max. fundamental cos φ active factor L2
         maxFundActiveFactorL3  : RealValueAndPNIOTimeStamp;   // Max. fundamental cos φ active factor L3
         maxTHDaNVoltL1  : RealValueAndPNIOTimeStamp;   // Max. THD+N voltage L1
         maxTHDaNVoltL2  : RealValueAndPNIOTimeStamp;   // Max. THD+N voltage L2
         maxTHDaNVoltL3  : RealValueAndPNIOTimeStamp;   // Max. THD+N voltage L3
         maxTHDaNCurrL1  : RealValueAndPNIOTimeStamp;   // Max. THD+N current L1
         maxTHDaNCurrL2  : RealValueAndPNIOTimeStamp;   // Max. THD+N current L2
         maxTHDaNCurrL3  : RealValueAndPNIOTimeStamp;   // Max. THD+N current L3
      END_STRUCT;
